LIN {X -0.159,Y -588.580,Z 1011.414,A 0.000,B 0.000,C 90.000,E1 110.536} C_DIS
LIN {X -0.262,Y -576.719,Z 1011.409,A 0.000,B 0.000,C 90.000,E1 109.577} C_DIS
LIN {X -0.071,Y -572.266,Z 1011.407,A 0.000,B 0.000,C 90.000,E1 109.214} C_DIS
LIN {X 0.230,Y -568.596,Z 1011.406,A 0.000,B 0.000,C 90.000,E1 108.960} C_DIS
LIN {X -0.107,Y -563.937,Z 1011.404,A 0.000,B 0.000,C 90.000,E1 108.725} C_DIS
LIN {X 0.068,Y -550.293,Z 1011.400,A 0.000,B 0.000,C 90.000,E1 108.000} C_DIS
LIN {X 0.171,Y -549.702,Z 1011.400,A 0.000,B 0.000,C 90.000,E1 107.946} C_DIS
LIN {X 0.114,Y -548.574,Z 1011.399,A 0.000,B 0.000,C 90.000,E1 107.819} C_DIS
LIN {X 0.072,Y -548.543,Z 1011.399,A 0.000,B 0.000,C 90.000,E1 107.819} C_DIS
LIN {X 0.076,Y -548.176,Z 1011.397,A 0.000,B 0.000,C 90.000,E1 107.511} C_DIS
LIN {X 0.119,Y -548.260,Z 1011.393,A 0.000,B 0.000,C 90.000,E1 106.804} C_DIS
LIN {X 0.030,Y -548.709,Z 1011.389,A 0.000,B 0.000,C 90.000,E1 105.969} C_DIS
LIN {X 0.074,Y -549.831,Z 1011.376,A 0.000,B 0.000,C 90.000,E1 103.716} C_DIS
LIN {X 0.056,Y -552.884,Z 1011.356,A 0.000,B 0.000,C 90.000,E1 100.074} C_DIS
LIN {X 0.060,Y -554.798,Z 1011.347,A 0.000,B 0.000,C 90.000,E1 98.398} C_DIS
LIN {X 0.114,Y -556.576,Z 1011.337,A 0.000,B 0.000,C 90.000,E1 96.720} C_DIS
LIN {X -0.128,Y -557.430,Z 1011.333,A 0.000,B 0.000,C 90.000,E1 95.910} C_DIS
LIN {X -0.220,Y -558.596,Z 1011.325,A 0.000,B 0.000,C 90.000,E1 94.531} C_DIS
LIN {X 0.262,Y -559.463,Z 1011.317,A 0.000,B 0.000,C 90.000,E1 93.094} C_DIS
LIN {X -0.033,Y -559.868,Z 1011.313,A 0.000,B 0.000,C 90.000,E1 92.293} C_DIS
LIN {X -0.023,Y -560.621,Z 1011.304,A 0.000,B 0.000,C 90.000,E1 90.630} C_DIS
LIN {X -0.009,Y -561.387,Z 1011.294,A 0.000,B 0.000,C 90.000,E1 88.969} C_DIS
LIN {X -0.164,Y -561.762,Z 1011.288,A 0.000,B 0.000,C 90.000,E1 87.879} C_DIS
LIN {X 0.253,Y -562.003,Z 1011.282,A 0.000,B 0.000,C 90.000,E1 86.731} C_DIS
LIN {X 0.100,Y -562.394,Z 1011.268,A 0.000,B 0.000,C 90.000,E1 84.261} C_DIS
LIN {X 0.005,Y -562.617,Z 1011.262,A 0.000,B 0.000,C 90.000,E1 83.166} C_DIS
LIN {X 0.214,Y -562.994,Z 1011.253,A 0.000,B 0.000,C 90.000,E1 81.489} C_DIS
LIN {X 0.027,Y -563.601,Z 1011.242,A 0.000,B 0.000,C 90.000,E1 79.577} C_DIS
LIN {X 0.059,Y -564.463,Z 1011.231,A 0.000,B 0.000,C 90.000,E1 77.645} C_DIS
LIN {X -0.086,Y -565.240,Z 1011.224,A 0.000,B 0.000,C 90.000,E1 76.284} C_DIS
LIN {X -0.261,Y -566.722,Z 1011.212,A 0.000,B 0.000,C 90.000,E1 74.102} C_DIS
LIN {X 0.119,Y -567.995,Z 1011.202,A 0.000,B 0.000,C 90.000,E1 72.417} C_DIS
LIN {X -0.006,Y -569.187,Z 1011.193,A 0.000,B 0.000,C 90.000,E1 70.786} C_DIS
LIN {X -0.082,Y -569.968,Z 1011.187,A 0.000,B 0.000,C 90.000,E1 69.699} C_DIS
LIN {X 0.010,Y -570.996,Z 1011.178,A 0.000,B 0.000,C 90.000,E1 68.050} C_DIS
LIN {X -0.367,Y -572.057,Z 1011.167,A 0.000,B 0.000,C 90.000,E1 66.177} C_DIS
LIN {X -0.319,Y -572.740,Z 1011.158,A 0.000,B 0.000,C 90.000,E1 64.537} C_DIS
LIN {X -0.007,Y -573.387,Z 1011.149,A 0.000,B 0.000,C 90.000,E1 62.871} C_DIS
LIN {X -0.193,Y -573.864,Z 1011.140,A 0.000,B 0.000,C 90.000,E1 61.257} C_DIS
LIN {X 0.064,Y -574.299,Z 1011.133,A 0.000,B 0.000,C 90.000,E1 59.871} C_DIS
LIN {X -0.165,Y -574.663,Z 1011.125,A 0.000,B 0.000,C 90.000,E1 58.535} C_DIS
LIN {X -0.083,Y -574.902,Z 1011.118,A 0.000,B 0.000,C 90.000,E1 57.168} C_DIS
LIN {X 0.005,Y -575.170,Z 1011.110,A 0.000,B 0.000,C 90.000,E1 55.801} C_DIS
LIN {X -0.384,Y -575.243,Z 1011.103,A 0.000,B 0.000,C 90.000,E1 54.482} C_DIS
LIN {X 0.216,Y -575.087,Z 1011.096,A 0.000,B 0.000,C 90.000,E1 53.336} C_DIS
LIN {X -0.140,Y -574.888,Z 1011.092,A 0.000,B 0.000,C 90.000,E1 52.557} C_DIS
LIN {X -0.001,Y -574.493,Z 1011.086,A 0.000,B 0.000,C 90.000,E1 51.457} C_DIS
LIN {X 0.134,Y -573.938,Z 1011.080,A 0.000,B 0.000,C 90.000,E1 50.356} C_DIS
LIN {X -0.182,Y -573.202,Z 1011.074,A 0.000,B 0.000,C 90.000,E1 49.299} C_DIS
LIN {X 0.300,Y -572.280,Z 1011.068,A 0.000,B 0.000,C 90.000,E1 48.162} C_DIS
LIN {X -0.167,Y -571.440,Z 1011.063,A 0.000,B 0.000,C 90.000,E1 47.391} C_DIS
LIN {X 0.162,Y -570.483,Z 1011.059,A 0.000,B 0.000,C 90.000,E1 46.539} C_DIS
LIN {X 0.368,Y -569.758,Z 1011.056,A 0.000,B 0.000,C 90.000,E1 45.972} C_DIS
LIN {X 0.056,Y -567.416,Z 1011.048,A 0.000,B 0.000,C 90.000,E1 44.636} C_DIS
LIN {X 0.021,Y -565.258,Z 1011.042,A 0.000,B 0.000,C 90.000,E1 43.542} C_DIS
LIN {X -0.198,Y -564.074,Z 1011.039,A 0.000,B 0.000,C 90.000,E1 43.014} C_DIS
LIN {X -0.271,Y -561.257,Z 1011.033,A 0.000,B 0.000,C 90.000,E1 41.919} C_DIS
LIN {X -0.140,Y -559.686,Z 1011.030,A 0.000,B 0.000,C 90.000,E1 41.353} C_DIS
LIN {X -0.309,Y -557.052,Z 1011.025,A 0.000,B 0.000,C 90.000,E1 40.539} C_DIS
LIN {X 0.281,Y -554.198,Z 1011.020,A 0.000,B 0.000,C 90.000,E1 39.644} C_DIS
LIN {X 0.060,Y -550.991,Z 1011.016,A 0.000,B 0.000,C 90.000,E1 38.830} C_DIS
LIN {X -0.196,Y -547.378,Z 1011.011,A 0.000,B 0.000,C 90.000,E1 38.016} C_DIS
LIN {X -0.064,Y -543.509,Z 1011.006,A 0.000,B 0.000,C 90.000,E1 37.156} C_DIS
LIN {X 0.045,Y -537.994,Z 1011.000,A 0.000,B 0.000,C 90.000,E1 36.011} C_DIS
LIN {X 0.068,Y -533.541,Z 1010.995,A 0.000,B 0.000,C 90.000,E1 35.152} C_DIS
LIN {X -0.247,Y -530.376,Z 1010.992,A 0.000,B 0.000,C 90.000,E1 34.612} C_DIS
LIN {X -0.037,Y -524.504,Z 1010.987,A 0.000,B 0.000,C 90.000,E1 33.579} C_DIS
LIN {X 0.150,Y -520.008,Z 1010.983,A 0.000,B 0.000,C 90.000,E1 32.832} C_DIS
LIN {X 0.030,Y -516.170,Z 1010.979,A 0.000,B 0.000,C 90.000,E1 32.260} C_DIS
LIN {X 0.042,Y -512.089,Z 1010.976,A 0.000,B 0.000,C 90.000,E1 31.671} C_DIS
LIN {X 0.030,Y -507.722,Z 1010.973,A 0.000,B 0.000,C 90.000,E1 31.082} C_DIS
LIN {X 0.054,Y -501.796,Z 1010.969,A 0.000,B 0.000,C 90.000,E1 30.335} C_DIS
LIN {X 0.046,Y -495.398,Z 1010.964,A 0.000,B 0.000,C 90.000,E1 29.589} C_DIS
LIN {X 0.004,Y -490.028,Z 1010.961,A 0.000,B 0.000,C 90.000,E1 28.999} C_DIS
LIN {X -0.134,Y -480.140,Z 1010.956,A 0.000,B 0.000,C 90.000,E1 28.025} C_DIS
LIN {X 0.044,Y -472.911,Z 1010.952,A 0.000,B 0.000,C 90.000,E1 27.308} C_DIS
LIN {X 0.131,Y -464.219,Z 1010.947,A 0.000,B 0.000,C 90.000,E1 26.488} C_DIS
LIN {X 0.025,Y -456.800,Z 1010.944,A 0.000,B 0.000,C 90.000,E1 25.848} C_DIS
LIN {X -0.094,Y -446.071,Z 1010.939,A 0.000,B 0.000,C 90.000,E1 24.951} C_DIS
LIN {X -0.172,Y -428.098,Z 1010.930,A 0.000,B 0.000,C 90.000,E1 23.387} C_DIS
LIN {X -0.101,Y -422.103,Z 1010.927,A 0.000,B 0.000,C 90.000,E1 22.823} C_DIS
LIN {X -0.068,Y -408.351,Z 1010.919,A 0.000,B 0.000,C 90.000,E1 21.408} C_DIS
LIN {X 0.103,Y -399.893,Z 1010.914,A 0.000,B 0.000,C 90.000,E1 20.429} C_DIS
LIN {X -0.029,Y -396.273,Z 1010.911,A 0.000,B 0.000,C 90.000,E1 19.993} C_DIS
LIN {X 0.148,Y -393.953,Z 1010.909,A 0.000,B 0.000,C 90.000,E1 19.577} C_DIS
LIN {X -0.191,Y -393.063,Z 1010.908,A 0.000,B 0.000,C 90.000,E1 19.450} C_DIS
LIN {X 0.130,Y -391.491,Z 1010.906,A 0.000,B 0.000,C 90.000,E1 18.960} C_DIS
LIN {X -0.058,Y -390.916,Z 1010.903,A 0.000,B 0.000,C 90.000,E1 18.544} C_DIS
LIN {X -0.011,Y -390.829,Z 1010.901,A 0.000,B 0.000,C 90.000,E1 18.181} C_DIS
LIN {X 0.033,Y -390.836,Z 1010.899,A 0.000,B 0.000,C 90.000,E1 17.819} C_DIS
LIN {X 0.185,Y -393.306,Z 1010.883,A 0.000,B 0.000,C 90.000,E1 14.954} C_DIS
LIN {X 0.162,Y -397.687,Z 1010.864,A 0.000,B 0.000,C 90.000,E1 11.422} C_DIS
LIN {X 0.087,Y -402.785,Z 1010.846,A 0.000,B 0.000,C 90.000,E1 8.276} C_DIS
LIN {X -0.040,Y -408.148,Z 1010.831,A 0.000,B 0.000,C 90.000,E1 5.511} C_DIS
LIN {X -0.042,Y -412.638,Z 1010.819,A 0.000,B 0.000,C 90.000,E1 3.440} C_DIS
LIN {X -0.010,Y -415.871,Z 1010.812,A 0.000,B 0.000,C 90.000,E1 2.064} C_DIS
LIN {X 0.024,Y -417.553,Z 1010.809,A 0.000,B 0.000,C 90.000,E1 1.547} C_DIS
LIN {X 0.134,Y -419.888,Z 1010.806,A 0.000,B 0.000,C 90.000,E1 1.031} C_DIS
LIN {X 0.165,Y -422.361,Z 1010.804,A 0.000,B 0.000,C 90.000,E1 0.688} C_DIS
LIN {X 0.184,Y -423.875,Z 1010.803,A 0.000,B 0.000,C 90.000,E1 0.516} C_DIS
LIN {X 0.059,Y -427.432,Z 1010.801,A 0.000,B 0.000,C 90.000,E1 0.229} C_DIS
LIN {X 0.165,Y -434.773,Z 1010.799,A 0.000,B 0.000,C 90.000,E1 359.771} C_DIS
LIN {X 0.007,Y -443.154,Z 1010.796,A 0.000,B 0.000,C 90.000,E1 359.312} C_DIS
LIN {X -0.039,Y -459.882,Z 1010.791,A 0.000,B 0.000,C 90.000,E1 358.339} C_DIS
LIN {X -0.089,Y -479.668,Z 1010.784,A 0.000,B 0.000,C 90.000,E1 357.192} C_DIS
LIN {X -0.222,Y -487.813,Z 1010.782,A 0.000,B 0.000,C 90.000,E1 356.731} C_DIS
LIN {X 0.114,Y -502.438,Z 1010.777,A 0.000,B 0.000,C 90.000,E1 355.812} C_DIS
LIN {X 0.211,Y -510.388,Z 1010.774,A 0.000,B 0.000,C 90.000,E1 355.298} C_DIS
LIN {X 0.103,Y -516.478,Z 1010.772,A 0.000,B 0.000,C 90.000,E1 354.894} C_DIS
LIN {X -0.247,Y -524.067,Z 1010.769,A 0.000,B 0.000,C 90.000,E1 354.375} C_DIS
LIN {X 0.169,Y -531.406,Z 1010.765,A 0.000,B 0.000,C 90.000,E1 353.742} C_DIS
LIN {X -0.197,Y -539.633,Z 1010.761,A 0.000,B 0.000,C 90.000,E1 353.053} C_DIS
LIN {X 0.217,Y -546.269,Z 1010.758,A 0.000,B 0.000,C 90.000,E1 352.356} C_DIS
LIN {X 0.030,Y -551.375,Z 1010.755,A 0.000,B 0.000,C 90.000,E1 351.837} C_DIS
LIN {X 0.311,Y -556.103,Z 1010.752,A 0.000,B 0.000,C 90.000,E1 351.254} C_DIS
LIN {X -0.315,Y -561.492,Z 1010.748,A 0.000,B 0.000,C 90.000,E1 350.622} C_DIS
LIN {X -0.010,Y -565.410,Z 1010.745,A 0.000,B 0.000,C 90.000,E1 350.038} C_DIS
LIN {X -0.230,Y -568.963,Z 1010.742,A 0.000,B 0.000,C 90.000,E1 349.511} C_DIS
LIN {X -0.145,Y -575.362,Z 1010.736,A 0.000,B 0.000,C 90.000,E1 348.409} C_DIS
LIN {X 0.154,Y -579.035,Z 1010.732,A 0.000,B 0.000,C 90.000,E1 347.701} C_DIS
LIN {X 0.260,Y -583.056,Z 1010.727,A 0.000,B 0.000,C 90.000,E1 346.881} C_DIS
LIN {X 0.082,Y -588.192,Z 1010.721,A 0.000,B 0.000,C 90.000,E1 345.825} C_DIS
LIN {X 0.347,Y -592.388,Z 1010.716,A 0.000,B 0.000,C 90.000,E1 344.866} C_DIS
LIN {X -0.133,Y -597.005,Z 1010.710,A 0.000,B 0.000,C 90.000,E1 343.850} C_DIS
LIN {X -0.266,Y -602.405,Z 1010.703,A 0.000,B 0.000,C 90.000,E1 342.543} C_DIS
LIN {X -0.138,Y -607.443,Z 1010.696,A 0.000,B 0.000,C 90.000,E1 341.221} C_DIS
LIN {X 0.025,Y -610.304,Z 1010.691,A 0.000,B 0.000,C 90.000,E1 340.423} C_DIS
LIN {X 0.012,Y -612.929,Z 1010.687,A 0.000,B 0.000,C 90.000,E1 339.645} C_DIS
LIN {X 0.167,Y -616.982,Z 1010.680,A 0.000,B 0.000,C 90.000,E1 338.337} C_DIS
LIN {X 0.156,Y -621.442,Z 1010.671,A 0.000,B 0.000,C 90.000,E1 336.794} C_DIS
LIN {X -0.107,Y -624.118,Z 1010.666,A 0.000,B 0.000,C 90.000,E1 335.793} C_DIS
LIN {X -0.339,Y -626.594,Z 1010.660,A 0.000,B 0.000,C 90.000,E1 334.793} C_DIS
LIN {X -0.250,Y -629.500,Z 1010.653,A 0.000,B 0.000,C 90.000,E1 333.512} C_DIS
LIN {X -0.171,Y -630.936,Z 1010.649,A 0.000,B 0.000,C 90.000,E1 332.743} C_DIS
LIN {X -0.048,Y -632.856,Z 1010.643,A 0.000,B 0.000,C 90.000,E1 331.719} C_DIS
LIN {X -0.077,Y -635.383,Z 1010.634,A 0.000,B 0.000,C 90.000,E1 330.205} C_DIS
LIN {X -0.185,Y -636.529,Z 1010.630,A 0.000,B 0.000,C 90.000,E1 329.459} C_DIS
LIN {X -0.189,Y -638.190,Z 1010.623,A 0.000,B 0.000,C 90.000,E1 328.201} C_DIS
LIN {X 0.125,Y -639.381,Z 1010.618,A 0.000,B 0.000,C 90.000,E1 327.168} C_DIS
LIN {X -0.031,Y -640.710,Z 1010.611,A 0.000,B 0.000,C 90.000,E1 325.928} C_DIS
LIN {X 0.319,Y -641.463,Z 1010.605,A 0.000,B 0.000,C 90.000,E1 324.895} C_DIS
LIN {X 0.152,Y -642.056,Z 1010.600,A 0.000,B 0.000,C 90.000,E1 323.909} C_DIS
LIN {X -0.116,Y -642.558,Z 1010.593,A 0.000,B 0.000,C 90.000,E1 322.683} C_DIS
LIN {X -0.052,Y -643.140,Z 1010.582,A 0.000,B 0.000,C 90.000,E1 320.678} C_DIS
LIN {X 0.171,Y -644.162,Z 1010.568,A 0.000,B 0.000,C 90.000,E1 318.162} C_DIS
LIN {X -0.161,Y -644.774,Z 1010.561,A 0.000,B 0.000,C 90.000,E1 316.944} C_DIS
LIN {X 0.333,Y -645.537,Z 1010.552,A 0.000,B 0.000,C 90.000,E1 315.405} C_DIS
LIN {X -0.197,Y -646.759,Z 1010.541,A 0.000,B 0.000,C 90.000,E1 313.461} C_DIS
LIN {X -0.050,Y -647.516,Z 1010.534,A 0.000,B 0.000,C 90.000,E1 312.204} C_DIS
LIN {X 0.031,Y -648.357,Z 1010.525,A 0.000,B 0.000,C 90.000,E1 310.458} C_DIS
LIN {X -0.215,Y -648.925,Z 1010.517,A 0.000,B 0.000,C 90.000,E1 308.991} C_DIS
LIN {X -0.049,Y -649.465,Z 1010.508,A 0.000,B 0.000,C 90.000,E1 307.488} C_DIS
LIN {X 0.314,Y -649.765,Z 1010.501,A 0.000,B 0.000,C 90.000,E1 306.217} C_DIS
LIN {X -0.218,Y -649.975,Z 1010.495,A 0.000,B 0.000,C 90.000,E1 305.025} C_DIS
LIN {X -0.056,Y -651.341,Z 1010.475,A 0.000,B 0.000,C 90.000,E1 301.544} C_DIS
LIN {X -0.005,Y -653.853,Z 1010.460,A 0.000,B 0.000,C 90.000,E1 298.821} C_DIS
LIN {X -0.152,Y -656.585,Z 1010.448,A 0.000,B 0.000,C 90.000,E1 296.616} C_DIS
LIN {X 0.326,Y -657.849,Z 1010.442,A 0.000,B 0.000,C 90.000,E1 295.591} C_DIS
LIN {X -0.058,Y -658.955,Z 1010.437,A 0.000,B 0.000,C 90.000,E1 294.643} C_DIS
LIN {X 0.172,Y -659.664,Z 1010.431,A 0.000,B 0.000,C 90.000,E1 293.643} C_DIS
LIN {X 0.162,Y -659.900,Z 1010.429,A 0.000,B 0.000,C 90.000,E1 293.153} C_DIS
LIN {X -0.204,Y -660.124,Z 1010.423,A 0.000,B 0.000,C 90.000,E1 292.206} C_DIS
LIN {X -0.208,Y -659.893,Z 1010.421,A 0.000,B 0.000,C 90.000,E1 291.716} C_DIS
LIN {X -0.089,Y -659.582,Z 1010.419,A 0.000,B 0.000,C 90.000,E1 291.461} C_DIS
LIN {X -0.095,Y -658.617,Z 1010.417,A 0.000,B 0.000,C 90.000,E1 290.972} C_DIS
LIN {X -0.216,Y -657.599,Z 1010.415,A 0.000,B 0.000,C 90.000,E1 290.737} C_DIS
LIN {X -0.230,Y -655.013,Z 1010.412,A 0.000,B 0.000,C 90.000,E1 290.248} C_DIS
LIN {X -0.181,Y -653.942,Z 1010.412,A 0.000,B 0.000,C 90.000,E1 290.120} C_DIS
LIN {X 0.247,Y -648.184,Z 1010.409,A 0.000,B 0.000,C 90.000,E1 289.631} C_DIS
LIN {X -0.342,Y -646.603,Z 1010.409,A 0.000,B 0.000,C 90.000,E1 289.577} C_DIS
LIN {X 0.314,Y -640.242,Z 1010.407,A 0.000,B 0.000,C 90.000,E1 289.141} C_DIS
LIN {X -0.269,Y -633.177,Z 1010.405,A 0.000,B 0.000,C 90.000,E1 288.852} C_DIS
LIN {X -0.152,Y -629.797,Z 1010.404,A 0.000,B 0.000,C 90.000,E1 288.652} C_DIS
LIN {X -0.201,Y -629.765,Z 1010.404,A 0.000,B 0.000,C 90.000,E1 288.652} C_DIS
LIN {X 0.325,Y -628.643,Z 1010.403,A 0.000,B 0.000,C 90.000,E1 288.417} C_DIS
LIN {X 0.281,Y -628.644,Z 1010.403,A 0.000,B 0.000,C 90.000,E1 288.417} C_DIS
LIN {X -0.188,Y -632.132,Z 1010.399,A 0.000,B 0.000,C 90.000,E1 287.873} C_DIS
LIN {X -0.039,Y -635.307,Z 1010.397,A 0.000,B 0.000,C 90.000,E1 287.402} C_DIS
LIN {X -0.219,Y -637.821,Z 1010.395,A 0.000,B 0.000,C 90.000,E1 287.040} C_DIS
LIN {X -0.216,Y -638.747,Z 1010.394,A 0.000,B 0.000,C 90.000,E1 286.913} C_DIS
LIN {X 0.071,Y -642.338,Z 1010.390,A 0.000,B 0.000,C 90.000,E1 286.260} C_DIS
LIN {X 0.080,Y -643.126,Z 1010.390,A 0.000,B 0.000,C 90.000,E1 286.134} C_DIS
LIN {X 0.244,Y -646.733,Z 1010.386,A 0.000,B 0.000,C 90.000,E1 285.371} C_DIS
LIN {X -0.039,Y -648.542,Z 1010.383,A 0.000,B 0.000,C 90.000,E1 284.898} C_DIS
LIN {X -0.148,Y -650.055,Z 1010.380,A 0.000,B 0.000,C 90.000,E1 284.411} C_DIS
LIN {X 0.348,Y -650.753,Z 1010.379,A 0.000,B 0.000,C 90.000,E1 284.120} C_DIS
LIN {X 0.088,Y -651.781,Z 1010.376,A 0.000,B 0.000,C 90.000,E1 283.647} C_DIS
LIN {X -0.165,Y -652.511,Z 1010.373,A 0.000,B 0.000,C 90.000,E1 283.175} C_DIS
LIN {X 0.098,Y -653.160,Z 1010.369,A 0.000,B 0.000,C 90.000,E1 282.411} C_DIS
LIN {X 0.233,Y -653.263,Z 1010.365,A 0.000,B 0.000,C 90.000,E1 281.658} C_DIS
LIN {X -0.012,Y -653.008,Z 1010.362,A 0.000,B 0.000,C 90.000,E1 281.186} C_DIS
LIN {X -0.263,Y -652.505,Z 1010.359,A 0.000,B 0.000,C 90.000,E1 280.715} C_DIS
LIN {X 0.005,Y -651.696,Z 1010.357,A 0.000,B 0.000,C 90.000,E1 280.197} C_DIS
LIN {X -0.258,Y -650.574,Z 1010.354,A 0.000,B 0.000,C 90.000,E1 279.726} C_DIS
LIN {X 0.140,Y -649.971,Z 1010.353,A 0.000,B 0.000,C 90.000,E1 279.443} C_DIS
LIN {X -0.137,Y -648.356,Z 1010.350,A 0.000,B 0.000,C 90.000,E1 278.973} C_DIS
LIN {X 0.113,Y -646.327,Z 1010.347,A 0.000,B 0.000,C 90.000,E1 278.454} C_DIS
LIN {X -0.285,Y -643.886,Z 1010.344,A 0.000,B 0.000,C 90.000,E1 277.992} C_DIS
LIN {X 0.191,Y -642.464,Z 1010.343,A 0.000,B 0.000,C 90.000,E1 277.701} C_DIS
LIN {X -0.234,Y -639.084,Z 1010.340,A 0.000,B 0.000,C 90.000,E1 277.239} C_DIS
LIN {X -0.045,Y -635.183,Z 1010.337,A 0.000,B 0.000,C 90.000,E1 276.720} C_DIS
LIN {X -0.006,Y -629.271,Z 1010.334,A 0.000,B 0.000,C 90.000,E1 276.087} C_DIS
LIN {X 0.272,Y -624.170,Z 1010.331,A 0.000,B 0.000,C 90.000,E1 275.568} C_DIS
LIN {X 0.152,Y -618.794,Z 1010.328,A 0.000,B 0.000,C 90.000,E1 275.106} C_DIS
LIN {X -0.288,Y -612.957,Z 1010.326,A 0.000,B 0.000,C 90.000,E1 274.702} C_DIS
LIN {X 0.233,Y -606.741,Z 1010.324,A 0.000,B 0.000,C 90.000,E1 274.245} C_DIS
LIN {X -0.111,Y -600.202,Z 1010.322,A 0.000,B 0.000,C 90.000,E1 273.898} C_DIS
LIN {X 0.097,Y -594.950,Z 1010.320,A 0.000,B 0.000,C 90.000,E1 273.612} C_DIS
LIN {X 0.213,Y -591.632,Z 1010.319,A 0.000,B 0.000,C 90.000,E1 273.440} C_DIS
LIN {X -0.276,Y -585.600,Z 1010.318,A 0.000,B 0.000,C 90.000,E1 273.269} C_DIS
LIN {X -0.195,Y -577.962,Z 1010.317,A 0.000,B 0.000,C 90.000,E1 273.037} C_DIS
LIN {X 0.186,Y -572.428,Z 1010.316,A 0.000,B 0.000,C 90.000,E1 272.865} C_DIS
LIN {X 0.157,Y -565.651,Z 1010.315,A 0.000,B 0.000,C 90.000,E1 272.751} C_DIS
LIN {X 0.189,Y -558.341,Z 1010.315,A 0.000,B 0.000,C 90.000,E1 272.694} C_DIS
LIN {X 0.139,Y -543.327,Z 1010.315,A 0.000,B 0.000,C 90.000,E1 272.694} C_DIS
LIN {X 0.079,Y -542.751,Z 1010.313,A 0.000,B 0.000,C 90.000,E1 272.407} C_DIS
LIN {X 0.216,Y -542.125,Z 1010.310,A 0.000,B 0.000,C 90.000,E1 271.835} C_DIS
LIN {X -0.132,Y -540.870,Z 1010.299,A 0.000,B 0.000,C 90.000,E1 269.885} C_DIS
LIN {X -0.025,Y -539.956,Z 1010.291,A 0.000,B 0.000,C 90.000,E1 268.453} C_DIS
LIN {X 0.045,Y -539.358,Z 1010.287,A 0.000,B 0.000,C 90.000,E1 267.593} C_DIS
LIN {X 0.186,Y -537.812,Z 1010.276,A 0.000,B 0.000,C 90.000,E1 265.584} C_DIS
LIN {X -0.203,Y -536.488,Z 1010.266,A 0.000,B 0.000,C 90.000,E1 263.913} C_DIS
LIN {X -0.072,Y -535.236,Z 1010.258,A 0.000,B 0.000,C 90.000,E1 262.470} C_DIS
LIN {X 0.027,Y -533.831,Z 1010.250,A 0.000,B 0.000,C 90.000,E1 261.027} C_DIS
LIN {X 0.220,Y -532.615,Z 1010.244,A 0.000,B 0.000,C 90.000,E1 259.859} C_DIS
LIN {X -0.066,Y -530.067,Z 1010.231,A 0.000,B 0.000,C 90.000,E1 257.589} C_DIS
LIN {X 0.218,Y -528.545,Z 1010.223,A 0.000,B 0.000,C 90.000,E1 256.117} C_DIS
LIN {X 0.134,Y -526.260,Z 1010.212,A 0.000,B 0.000,C 90.000,E1 254.102} C_DIS
LIN {X -0.028,Y -524.699,Z 1010.204,A 0.000,B 0.000,C 90.000,E1 252.670} C_DIS
LIN {X -0.060,Y -523.087,Z 1010.196,A 0.000,B 0.000,C 90.000,E1 251.221} C_DIS
LIN {X 0.054,Y -521.211,Z 1010.188,A 0.000,B 0.000,C 90.000,E1 249.752} C_DIS
LIN {X -0.054,Y -518.588,Z 1010.176,A 0.000,B 0.000,C 90.000,E1 247.720} C_DIS
LIN {X 0.036,Y -516.984,Z 1010.170,A 0.000,B 0.000,C 90.000,E1 246.538} C_DIS
LIN {X -0.244,Y -514.866,Z 1010.162,A 0.000,B 0.000,C 90.000,E1 245.101} C_DIS
LIN {X -0.121,Y -513.572,Z 1010.157,A 0.000,B 0.000,C 90.000,E1 244.204} C_DIS
LIN {X -0.250,Y -511.196,Z 1010.148,A 0.000,B 0.000,C 90.000,E1 242.743} C_DIS
LIN {X 0.132,Y -508.341,Z 1010.139,A 0.000,B 0.000,C 90.000,E1 240.923} C_DIS
LIN {X -0.064,Y -505.758,Z 1010.130,A 0.000,B 0.000,C 90.000,E1 239.459} C_DIS
LIN {X 0.194,Y -504.107,Z 1010.125,A 0.000,B 0.000,C 90.000,E1 238.535} C_DIS
LIN {X 0.181,Y -501.177,Z 1010.117,A 0.000,B 0.000,C 90.000,E1 237.041} C_DIS
LIN {X -0.175,Y -498.568,Z 1010.110,A 0.000,B 0.000,C 90.000,E1 235.881} C_DIS
LIN {X -0.156,Y -496.584,Z 1010.105,A 0.000,B 0.000,C 90.000,E1 234.975} C_DIS
LIN {X -0.008,Y -493.625,Z 1010.099,A 0.000,B 0.000,C 90.000,E1 233.749} C_DIS
LIN {X -0.196,Y -490.682,Z 1010.092,A 0.000,B 0.000,C 90.000,E1 232.557} C_DIS
LIN {X -0.022,Y -485.613,Z 1010.080,A 0.000,B 0.000,C 90.000,E1 230.400} C_DIS
LIN {X 0.081,Y -482.059,Z 1010.072,A 0.000,B 0.000,C 90.000,E1 228.852} C_DIS
LIN {X 0.195,Y -475.944,Z 1010.056,A 0.000,B 0.000,C 90.000,E1 226.053} C_DIS
LIN {X 0.235,Y -471.520,Z 1010.044,A 0.000,B 0.000,C 90.000,E1 223.866} C_DIS
LIN {X 0.166,Y -466.861,Z 1010.032,A 0.000,B 0.000,C 90.000,E1 221.676} C_DIS
LIN {X 0.211,Y -463.462,Z 1010.023,A 0.000,B 0.000,C 90.000,E1 220.092} C_DIS
LIN {X 0.153,Y -460.594,Z 1010.016,A 0.000,B 0.000,C 90.000,E1 218.830} C_DIS
LIN {X -0.119,Y -456.352,Z 1010.005,A 0.000,B 0.000,C 90.000,E1 216.950} C_DIS
LIN {X -0.124,Y -452.141,Z 1009.995,A 0.000,B 0.000,C 90.000,E1 215.025} C_DIS
LIN {X 0.025,Y -446.480,Z 1009.980,A 0.000,B 0.000,C 90.000,E1 212.418} C_DIS
LIN {X 0.081,Y -441.507,Z 1009.967,A 0.000,B 0.000,C 90.000,E1 210.129} C_DIS
LIN {X 0.006,Y -439.348,Z 1009.962,A 0.000,B 0.000,C 90.000,E1 209.155} C_DIS
LIN {X -0.012,Y -434.779,Z 1009.951,A 0.000,B 0.000,C 90.000,E1 207.180} C_DIS
LIN {X -0.151,Y -431.069,Z 1009.942,A 0.000,B 0.000,C 90.000,E1 205.540} C_DIS
LIN {X 0.213,Y -427.325,Z 1009.933,A 0.000,B 0.000,C 90.000,E1 203.823} C_DIS
LIN {X 0.126,Y -422.103,Z 1009.919,A 0.000,B 0.000,C 90.000,E1 201.482} C_DIS
LIN {X -0.100,Y -417.314,Z 1009.906,A 0.000,B 0.000,C 90.000,E1 199.141} C_DIS
LIN {X 0.044,Y -412.927,Z 1009.893,A 0.000,B 0.000,C 90.000,E1 196.732} C_DIS
LIN {X -0.168,Y -408.922,Z 1009.880,A 0.000,B 0.000,C 90.000,E1 194.356} C_DIS
LIN {X 0.114,Y -405.296,Z 1009.866,A 0.000,B 0.000,C 90.000,E1 191.895} C_DIS
LIN {X -0.172,Y -402.664,Z 1009.855,A 0.000,B 0.000,C 90.000,E1 189.849} C_DIS
LIN {X -0.174,Y -402.053,Z 1009.851,A 0.000,B 0.000,C 90.000,E1 189.151} C_DIS
LIN {X -0.182,Y -401.886,Z 1009.847,A 0.000,B 0.000,C 90.000,E1 188.454} C_DIS
LIN {X -0.194,Y -402.215,Z 1009.843,A 0.000,B 0.000,C 90.000,E1 187.757} C_DIS
LIN {X 0.141,Y -403.219,Z 1009.839,A 0.000,B 0.000,C 90.000,E1 187.011} C_DIS
LIN {X 0.159,Y -404.411,Z 1009.836,A 0.000,B 0.000,C 90.000,E1 186.486} C_DIS
LIN {X -0.152,Y -407.346,Z 1009.832,A 0.000,B 0.000,C 90.000,E1 185.796} C_DIS
LIN {X -0.146,Y -409.187,Z 1009.830,A 0.000,B 0.000,C 90.000,E1 185.448} C_DIS
LIN {X -0.180,Y -412.261,Z 1009.827,A 0.000,B 0.000,C 90.000,E1 184.935} C_DIS
LIN {X 0.187,Y -415.702,Z 1009.825,A 0.000,B 0.000,C 90.000,E1 184.416} C_DIS
LIN {X 0.200,Y -428.181,Z 1009.816,A 0.000,B 0.000,C 90.000,E1 182.922} C_DIS
LIN {X 0.012,Y -436.600,Z 1009.811,A 0.000,B 0.000,C 90.000,E1 182.007} C_DIS
LIN {X -0.167,Y -446.138,Z 1009.805,A 0.000,B 0.000,C 90.000,E1 180.917} C_DIS
LIN {X 0.161,Y -455.560,Z 1009.799,A 0.000,B 0.000,C 90.000,E1 179.771} C_DIS
LIN {X 0.088,Y -463.361,Z 1009.794,A 0.000,B 0.000,C 90.000,E1 178.854} C_DIS
LIN {X 0.202,Y -469.855,Z 1009.789,A 0.000,B 0.000,C 90.000,E1 178.051} C_DIS
LIN {X 0.146,Y -478.630,Z 1009.783,A 0.000,B 0.000,C 90.000,E1 176.963} C_DIS
LIN {X -0.226,Y -482.138,Z 1009.781,A 0.000,B 0.000,C 90.000,E1 176.560} C_DIS
LIN {X -0.092,Y -486.756,Z 1009.777,A 0.000,B 0.000,C 90.000,E1 175.927} C_DIS
LIN {X -0.246,Y -495.535,Z 1009.771,A 0.000,B 0.000,C 90.000,E1 174.723} C_DIS
LIN {X -0.055,Y -503.529,Z 1009.764,A 0.000,B 0.000,C 90.000,E1 173.514} C_DIS
LIN {X -0.249,Y -511.268,Z 1009.757,A 0.000,B 0.000,C 90.000,E1 172.356} C_DIS
LIN {X -0.138,Y -517.755,Z 1009.752,A 0.000,B 0.000,C 90.000,E1 171.319} C_DIS
LIN {X 0.072,Y -527.246,Z 1009.743,A 0.000,B 0.000,C 90.000,E1 169.690} C_DIS
LIN {X 0.142,Y -536.544,Z 1009.734,A 0.000,B 0.000,C 90.000,E1 168.117} C_DIS
LIN {X -0.093,Y -545.559,Z 1009.725,A 0.000,B 0.000,C 90.000,E1 166.589} C_DIS
LIN {X 0.262,Y -555.100,Z 1009.716,A 0.000,B 0.000,C 90.000,E1 164.866} C_DIS
LIN {X -0.023,Y -560.425,Z 1009.711,A 0.000,B 0.000,C 90.000,E1 163.921} C_DIS
LIN {X -0.204,Y -566.237,Z 1009.705,A 0.000,B 0.000,C 90.000,E1 162.834} C_DIS
LIN {X 0.066,Y -571.839,Z 1009.698,A 0.000,B 0.000,C 90.000,E1 161.710} C_DIS
LIN {X -0.137,Y -575.954,Z 1009.694,A 0.000,B 0.000,C 90.000,E1 160.913} C_DIS
LIN {X -0.182,Y -581.717,Z 1009.687,A 0.000,B 0.000,C 90.000,E1 159.699} C_DIS
LIN {X 0.133,Y -586.580,Z 1009.681,A 0.000,B 0.000,C 90.000,E1 158.592} C_DIS
LIN {X -0.034,Y -591.112,Z 1009.675,A 0.000,B 0.000,C 90.000,E1 157.539} C_DIS
LIN {X -0.143,Y -595.323,Z 1009.669,A 0.000,B 0.000,C 90.000,E1 156.485} C_DIS
LIN {X 0.218,Y -597.338,Z 1009.666,A 0.000,B 0.000,C 90.000,E1 155.921} C_DIS
LIN {X -0.106,Y -600.991,Z 1009.661,A 0.000,B 0.000,C 90.000,E1 154.897} C_DIS
LIN {X -0.097,Y -604.322,Z 1009.655,A 0.000,B 0.000,C 90.000,E1 153.845} C_DIS
LIN {X -0.053,Y -607.431,Z 1009.649,A 0.000,B 0.000,C 90.000,E1 152.794} C_DIS
LIN {X -0.322,Y -611.868,Z 1009.640,A 0.000,B 0.000,C 90.000,E1 151.257} C_DIS
LIN {X -0.167,Y -614.725,Z 1009.634,A 0.000,B 0.000,C 90.000,E1 150.205} C_DIS
LIN {X -0.233,Y -618.884,Z 1009.626,A 0.000,B 0.000,C 90.000,E1 148.663} C_DIS
LIN {X -0.216,Y -622.939,Z 1009.617,A 0.000,B 0.000,C 90.000,E1 147.120} C_DIS
LIN {X 0.041,Y -627.626,Z 1009.607,A 0.000,B 0.000,C 90.000,E1 145.308} C_DIS
LIN {X 0.050,Y -631.630,Z 1009.599,A 0.000,B 0.000,C 90.000,E1 143.783} C_DIS
LIN {X -0.383,Y -634.920,Z 1009.592,A 0.000,B 0.000,C 90.000,E1 142.557} C_DIS
LIN {X 0.024,Y -638.840,Z 1009.583,A 0.000,B 0.000,C 90.000,E1 141.009} C_DIS
LIN {X 0.026,Y -642.641,Z 1009.575,A 0.000,B 0.000,C 90.000,E1 139.504} C_DIS
LIN {X 0.249,Y -645.132,Z 1009.570,A 0.000,B 0.000,C 90.000,E1 138.485} C_DIS
LIN {X -0.034,Y -647.664,Z 1009.564,A 0.000,B 0.000,C 90.000,E1 137.514} C_DIS
LIN {X -0.033,Y -653.693,Z 1009.552,A 0.000,B 0.000,C 90.000,E1 135.283} C_DIS
LIN {X -0.353,Y -661.246,Z 1009.538,A 0.000,B 0.000,C 90.000,E1 132.852} C_DIS
LIN {X 0.037,Y -666.002,Z 1009.530,A 0.000,B 0.000,C 90.000,E1 131.353} C_DIS
LIN {X 0.148,Y -670.627,Z 1009.522,A 0.000,B 0.000,C 90.000,E1 129.886} C_DIS
LIN {X 0.256,Y -674.200,Z 1009.515,A 0.000,B 0.000,C 90.000,E1 128.669} C_DIS
LIN {X -0.429,Y -677.664,Z 1009.508,A 0.000,B 0.000,C 90.000,E1 127.523} C_DIS
LIN {X -0.106,Y -680.995,Z 1009.502,A 0.000,B 0.000,C 90.000,E1 126.297} C_DIS
LIN {X -0.121,Y -684.893,Z 1009.494,A 0.000,B 0.000,C 90.000,E1 124.865} C_DIS
LIN {X -0.108,Y -687.414,Z 1009.488,A 0.000,B 0.000,C 90.000,E1 123.913} C_DIS
LIN {X 0.312,Y -689.241,Z 1009.484,A 0.000,B 0.000,C 90.000,E1 123.166} C_DIS
LIN {X -0.095,Y -693.402,Z 1009.475,A 0.000,B 0.000,C 90.000,E1 121.544} C_DIS
LIN {X 0.033,Y -695.735,Z 1009.470,A 0.000,B 0.000,C 90.000,E1 120.590} C_DIS
LIN {X -0.169,Y -697.719,Z 1009.465,A 0.000,B 0.000,C 90.000,E1 119.667} C_DIS
LIN {X 0.266,Y -699.301,Z 1009.460,A 0.000,B 0.000,C 90.000,E1 118.693} C_DIS
LIN {X -0.164,Y -700.269,Z 1009.456,A 0.000,B 0.000,C 90.000,E1 118.025} C_DIS
LIN {X 0.378,Y -700.744,Z 1009.453,A 0.000,B 0.000,C 90.000,E1 117.513} C_DIS
LIN {X 0.077,Y -702.241,Z 1009.443,A 0.000,B 0.000,C 90.000,E1 115.668} C_DIS
LIN {X -0.376,Y -702.886,Z 1009.438,A 0.000,B 0.000,C 90.000,E1 114.771} C_DIS
LIN {X 0.182,Y -702.947,Z 1009.435,A 0.000,B 0.000,C 90.000,E1 114.259} C_DIS
LIN {X 0.173,Y -702.802,Z 1009.434,A 0.000,B 0.000,C 90.000,E1 114.027} C_DIS
LIN {X 0.085,Y -702.062,Z 1009.431,A 0.000,B 0.000,C 90.000,E1 113.567} C_DIS
LIN {X 0.081,Y -701.260,Z 1009.430,A 0.000,B 0.000,C 90.000,E1 113.334} C_DIS
LIN {X 0.353,Y -700.222,Z 1009.428,A 0.000,B 0.000,C 90.000,E1 113.078} C_DIS
LIN {X -0.295,Y -699.036,Z 1009.427,A 0.000,B 0.000,C 90.000,E1 112.898} C_DIS
LIN {X -0.162,Y -698.192,Z 1009.426,A 0.000,B 0.000,C 90.000,E1 112.770} C_DIS
LIN {X -0.030,Y -696.938,Z 1009.426,A 0.000,B 0.000,C 90.000,E1 112.642} C_DIS
LIN {X 0.187,Y -690.637,Z 1009.424,A 0.000,B 0.000,C 90.000,E1 112.206} C_DIS
LIN {X -0.300,Y -688.644,Z 1009.423,A 0.000,B 0.000,C 90.000,E1 112.153} C_DIS
LIN {X 0.064,Y -683.849,Z 1009.422,A 0.000,B 0.000,C 90.000,E1 111.972} C_DIS
LIN {X 0.183,Y -675.272,Z 1009.422,A 0.000,B 0.000,C 90.000,E1 111.844} C_DIS
LIN {X 0.132,Y -617.756,Z 1009.421,A 0.000,B 0.000,C 90.000,E1 111.844} C_DIS
LIN {X 0.110,Y -610.545,Z 1009.420,A 0.000,B 0.000,C 90.000,E1 111.663} C_DIS
LIN {X 0.263,Y -605.563,Z 1009.419,A 0.000,B 0.000,C 90.000,E1 111.461} C_DIS
LIN {X 0.108,Y -599.880,Z 1009.418,A 0.000,B 0.000,C 90.000,E1 111.227} C_DIS
LIN {X 0.042,Y -593.741,Z 1009.416,A 0.000,B 0.000,C 90.000,E1 110.865} C_DIS
LIN {X -0.211,Y -588.092,Z 1009.414,A 0.000,B 0.000,C 90.000,E1 110.482} C_DIS
LIN {X -0.126,Y -577.105,Z 1009.409,A 0.000,B 0.000,C 90.000,E1 109.577} C_DIS
LIN {X 0.078,Y -572.714,Z 1009.407,A 0.000,B 0.000,C 90.000,E1 109.214} C_DIS
LIN {X 0.217,Y -571.073,Z 1009.406,A 0.000,B 0.000,C 90.000,E1 109.087} C_DIS
LIN {X 0.014,Y -564.479,Z 1009.404,A 0.000,B 0.000,C 90.000,E1 108.725} C_DIS
LIN {X -0.112,Y -550.170,Z 1009.400,A 0.000,B 0.000,C 90.000,E1 108.000} C_DIS
LIN {X 0.003,Y -548.609,Z 1009.399,A 0.000,B 0.000,C 90.000,E1 107.819} C_DIS
LIN {X -0.039,Y -548.604,Z 1009.399,A 0.000,B 0.000,C 90.000,E1 107.819} C_DIS
LIN {X 0.134,Y -548.234,Z 1009.397,A 0.000,B 0.000,C 90.000,E1 107.511} C_DIS
LIN {X -0.100,Y -548.456,Z 1009.392,A 0.000,B 0.000,C 90.000,E1 106.551} C_DIS
LIN {X -0.096,Y -548.996,Z 1009.386,A 0.000,B 0.000,C 90.000,E1 105.426} C_DIS
LIN {X -0.164,Y -550.041,Z 1009.375,A 0.000,B 0.000,C 90.000,E1 103.467} C_DIS
LIN {X 0.142,Y -553.225,Z 1009.355,A 0.000,B 0.000,C 90.000,E1 99.792} C_DIS
LIN {X 0.247,Y -555.100,Z 1009.345,A 0.000,B 0.000,C 90.000,E1 98.106} C_DIS
LIN {X 0.177,Y -556.575,Z 1009.337,A 0.000,B 0.000,C 90.000,E1 96.720} C_DIS
LIN {X -0.064,Y -557.454,Z 1009.333,A 0.000,B 0.000,C 90.000,E1 95.910} C_DIS
LIN {X -0.157,Y -558.592,Z 1009.325,A 0.000,B 0.000,C 90.000,E1 94.531} C_DIS
LIN {X -0.233,Y -559.459,Z 1009.317,A 0.000,B 0.000,C 90.000,E1 93.151} C_DIS
LIN {X 0.030,Y -559.865,Z 1009.313,A 0.000,B 0.000,C 90.000,E1 92.293} C_DIS
LIN {X 0.135,Y -560.766,Z 1009.302,A 0.000,B 0.000,C 90.000,E1 90.344} C_DIS
LIN {X 0.055,Y -561.416,Z 1009.294,A 0.000,B 0.000,C 90.000,E1 88.969} C_DIS
LIN {X -0.100,Y -561.793,Z 1009.288,A 0.000,B 0.000,C 90.000,E1 87.879} C_DIS
LIN {X -0.147,Y -562.036,Z 1009.281,A 0.000,B 0.000,C 90.000,E1 86.502} C_DIS
LIN {X 0.165,Y -562.393,Z 1009.268,A 0.000,B 0.000,C 90.000,E1 84.261} C_DIS
LIN {X 0.220,Y -562.598,Z 1009.261,A 0.000,B 0.000,C 90.000,E1 82.875} C_DIS
LIN {X -0.121,Y -563.047,Z 1009.251,A 0.000,B 0.000,C 90.000,E1 81.254} C_DIS
LIN {X -0.302,Y -563.693,Z 1009.241,A 0.000,B 0.000,C 90.000,E1 79.342} C_DIS
LIN {X 0.064,Y -564.925,Z 1009.227,A 0.000,B 0.000,C 90.000,E1 76.825} C_DIS
LIN {X 0.021,Y -566.297,Z 1009.215,A 0.000,B 0.000,C 90.000,E1 74.629} C_DIS
LIN {X 0.232,Y -567.548,Z 1009.206,A 0.000,B 0.000,C 90.000,E1 72.960} C_DIS
LIN {X -0.243,Y -568.561,Z 1009.198,A 0.000,B 0.000,C 90.000,E1 71.638} C_DIS
LIN {X 0.170,Y -569.782,Z 1009.189,A 0.000,B 0.000,C 90.000,E1 69.953} C_DIS
LIN {X 0.073,Y -570.948,Z 1009.178,A 0.000,B 0.000,C 90.000,E1 68.050} C_DIS
LIN {X -0.306,Y -571.990,Z 1009.168,A 0.000,B 0.000,C 90.000,E1 66.177} C_DIS
LIN {X -0.259,Y -572.666,Z 1009.158,A 0.000,B 0.000,C 90.000,E1 64.537} C_DIS
LIN {X 0.051,Y -573.286,Z 1009.149,A 0.000,B 0.000,C 90.000,E1 62.871} C_DIS
LIN {X -0.137,Y -573.768,Z 1009.140,A 0.000,B 0.000,C 90.000,E1 61.257} C_DIS
LIN {X 0.118,Y -574.205,Z 1009.133,A 0.000,B 0.000,C 90.000,E1 59.871} C_DIS
LIN {X -0.113,Y -574.537,Z 1009.125,A 0.000,B 0.000,C 90.000,E1 58.535} C_DIS
LIN {X -0.174,Y -574.711,Z 1009.119,A 0.000,B 0.000,C 90.000,E1 57.454} C_DIS
LIN {X -0.092,Y -574.962,Z 1009.112,A 0.000,B 0.000,C 90.000,E1 56.087} C_DIS
LIN {X 0.167,Y -575.067,Z 1009.106,A 0.000,B 0.000,C 90.000,E1 54.975} C_DIS
LIN {X -0.041,Y -575.006,Z 1009.100,A 0.000,B 0.000,C 90.000,E1 53.909} C_DIS
LIN {X -0.248,Y -574.837,Z 1009.094,A 0.000,B 0.000,C 90.000,E1 52.844} C_DIS
LIN {X 0.038,Y -574.314,Z 1009.086,A 0.000,B 0.000,C 90.000,E1 51.457} C_DIS
LIN {X 0.170,Y -573.733,Z 1009.080,A 0.000,B 0.000,C 90.000,E1 50.356} C_DIS
LIN {X -0.148,Y -572.982,Z 1009.074,A 0.000,B 0.000,C 90.000,E1 49.299} C_DIS
LIN {X 0.331,Y -572.051,Z 1009.068,A 0.000,B 0.000,C 90.000,E1 48.162} C_DIS
LIN {X -0.139,Y -571.192,Z 1009.063,A 0.000,B 0.000,C 90.000,E1 47.391} C_DIS
LIN {X 0.186,Y -570.209,Z 1009.059,A 0.000,B 0.000,C 90.000,E1 46.539} C_DIS
LIN {X 0.391,Y -569.455,Z 1009.056,A 0.000,B 0.000,C 90.000,E1 45.972} C_DIS
LIN {X -0.018,Y -567.552,Z 1009.050,A 0.000,B 0.000,C 90.000,E1 44.919} C_DIS
LIN {X 0.347,Y -565.476,Z 1009.044,A 0.000,B 0.000,C 90.000,E1 43.785} C_DIS
LIN {X -0.188,Y -563.681,Z 1009.039,A 0.000,B 0.000,C 90.000,E1 43.014} C_DIS
LIN {X -0.268,Y -560.843,Z 1009.033,A 0.000,B 0.000,C 90.000,E1 41.919} C_DIS
LIN {X -0.138,Y -559.210,Z 1009.030,A 0.000,B 0.000,C 90.000,E1 41.353} C_DIS
LIN {X -0.312,Y -556.562,Z 1009.025,A 0.000,B 0.000,C 90.000,E1 40.539} C_DIS
LIN {X 0.273,Y -553.669,Z 1009.020,A 0.000,B 0.000,C 90.000,E1 39.644} C_DIS
LIN {X 0.045,Y -550.350,Z 1009.016,A 0.000,B 0.000,C 90.000,E1 38.830} C_DIS
LIN {X -0.026,Y -546.107,Z 1009.010,A 0.000,B 0.000,C 90.000,E1 37.855} C_DIS
LIN {X 0.087,Y -542.114,Z 1009.006,A 0.000,B 0.000,C 90.000,E1 36.996} C_DIS
LIN {X -0.010,Y -538.616,Z 1009.002,A 0.000,B 0.000,C 90.000,E1 36.297} C_DIS
LIN {X 0.023,Y -534.258,Z 1008.997,A 0.000,B 0.000,C 90.000,E1 35.438} C_DIS
LIN {X -0.298,Y -529.525,Z 1008.992,A 0.000,B 0.000,C 90.000,E1 34.612} C_DIS
LIN {X 0.065,Y -524.463,Z 1008.987,A 0.000,B 0.000,C 90.000,E1 33.706} C_DIS
LIN {X 0.080,Y -519.053,Z 1008.982,A 0.000,B 0.000,C 90.000,E1 32.832} C_DIS
LIN {X -0.045,Y -515.158,Z 1008.979,A 0.000,B 0.000,C 90.000,E1 32.260} C_DIS
LIN {X -0.041,Y -511.031,Z 1008.976,A 0.000,B 0.000,C 90.000,E1 31.671} C_DIS
LIN {X 0.121,Y -507.755,Z 1008.974,A 0.000,B 0.000,C 90.000,E1 31.209} C_DIS
LIN {X 0.077,Y -503.036,Z 1008.970,A 0.000,B 0.000,C 90.000,E1 30.620} C_DIS
LIN {X 0.253,Y -498.033,Z 1008.967,A 0.000,B 0.000,C 90.000,E1 30.001} C_DIS
LIN {X 0.012,Y -491.473,Z 1008.963,A 0.000,B 0.000,C 90.000,E1 29.283} C_DIS
LIN {X 0.125,Y -484.556,Z 1008.959,A 0.000,B 0.000,C 90.000,E1 28.565} C_DIS
LIN {X -0.006,Y -476.375,Z 1008.954,A 0.000,B 0.000,C 90.000,E1 27.769} C_DIS
LIN {X -0.072,Y -467.597,Z 1008.950,A 0.000,B 0.000,C 90.000,E1 26.950} C_DIS
LIN {X 0.239,Y -458.643,Z 1008.945,A 0.000,B 0.000,C 90.000,E1 26.104} C_DIS
LIN {X 0.095,Y -447.906,Z 1008.940,A 0.000,B 0.000,C 90.000,E1 25.207} C_DIS
LIN {X 0.161,Y -422.477,Z 1008.928,A 0.000,B 0.000,C 90.000,E1 22.950} C_DIS
LIN {X -0.089,Y -408.320,Z 1008.920,A 0.000,B 0.000,C 90.000,E1 21.535} C_DIS
LIN {X -0.158,Y -399.958,Z 1008.914,A 0.000,B 0.000,C 90.000,E1 20.610} C_DIS
LIN {X 0.111,Y -395.987,Z 1008.912,A 0.000,B 0.000,C 90.000,E1 20.066} C_DIS
LIN {X 0.039,Y -393.076,Z 1008.909,A 0.000,B 0.000,C 90.000,E1 19.577} C_DIS
LIN {X -0.186,Y -391.217,Z 1008.906,A 0.000,B 0.000,C 90.000,E1 19.033} C_DIS
LIN {X -0.179,Y -390.736,Z 1008.903,A 0.000,B 0.000,C 90.000,E1 18.544} C_DIS
LIN {X -0.155,Y -390.669,Z 1008.902,A 0.000,B 0.000,C 90.000,E1 18.362} C_DIS
LIN {X -0.127,Y -390.799,Z 1008.899,A 0.000,B 0.000,C 90.000,E1 17.819} C_DIS
LIN {X 0.032,Y -395.041,Z 1008.875,A 0.000,B 0.000,C 90.000,E1 13.536} C_DIS
LIN {X -0.061,Y -402.302,Z 1008.848,A 0.000,B 0.000,C 90.000,E1 8.624} C_DIS
LIN {X -0.194,Y -408.283,Z 1008.831,A 0.000,B 0.000,C 90.000,E1 5.511} C_DIS
LIN {X -0.188,Y -412.021,Z 1008.821,A 0.000,B 0.000,C 90.000,E1 3.784} C_DIS
LIN {X -0.170,Y -415.081,Z 1008.813,A 0.000,B 0.000,C 90.000,E1 2.407} C_DIS
LIN {X -0.135,Y -416.946,Z 1008.810,A 0.000,B 0.000,C 90.000,E1 1.718} C_DIS
LIN {X -0.109,Y -419.071,Z 1008.807,A 0.000,B 0.000,C 90.000,E1 1.203} C_DIS
LIN {X -0.097,Y -419.896,Z 1008.806,A 0.000,B 0.000,C 90.000,E1 1.031} C_DIS
LIN {X 0.153,Y -422.853,Z 1008.803,A 0.000,B 0.000,C 90.000,E1 0.573} C_DIS
LIN {X -0.030,Y -425.482,Z 1008.802,A 0.000,B 0.000,C 90.000,E1 0.344} C_DIS
LIN {X -0.211,Y -427.044,Z 1008.801,A 0.000,B 0.000,C 90.000,E1 0.229} C_DIS
LIN {X 0.000,Y -430.047,Z 1008.800,A 0.000,B 0.000,C 90.000,E1 360.000} C_DIS
LIN {X -0.082,Y -437.099,Z 1008.798,A 0.000,B 0.000,C 90.000,E1 359.599} C_DIS
LIN {X 0.078,Y -443.801,Z 1008.796,A 0.000,B 0.000,C 90.000,E1 359.198} C_DIS
LIN {X 0.182,Y -460.297,Z 1008.790,A 0.000,B 0.000,C 90.000,E1 358.224} C_DIS
LIN {X -0.199,Y -476.871,Z 1008.785,A 0.000,B 0.000,C 90.000,E1 357.306} C_DIS
LIN {X -0.138,Y -486.621,Z 1008.782,A 0.000,B 0.000,C 90.000,E1 356.731} C_DIS
LIN {X -0.234,Y -496.436,Z 1008.779,A 0.000,B 0.000,C 90.000,E1 356.159} C_DIS
LIN {X 0.138,Y -506.063,Z 1008.775,A 0.000,B 0.000,C 90.000,E1 355.527} C_DIS
LIN {X 0.135,Y -512.346,Z 1008.773,A 0.000,B 0.000,C 90.000,E1 355.122} C_DIS
LIN {X -0.130,Y -518.470,Z 1008.771,A 0.000,B 0.000,C 90.000,E1 354.723} C_DIS
LIN {X 0.003,Y -524.519,Z 1008.768,A 0.000,B 0.000,C 90.000,E1 354.261} C_DIS
LIN {X -0.073,Y -531.811,Z 1008.765,A 0.000,B 0.000,C 90.000,E1 353.685} C_DIS
LIN {X 0.138,Y -538.757,Z 1008.762,A 0.000,B 0.000,C 90.000,E1 353.053} C_DIS
LIN {X 0.179,Y -544.192,Z 1008.759,A 0.000,B 0.000,C 90.000,E1 352.534} C_DIS
LIN {X -0.065,Y -550.563,Z 1008.755,A 0.000,B 0.000,C 90.000,E1 351.894} C_DIS
LIN {X 0.188,Y -555.371,Z 1008.752,A 0.000,B 0.000,C 90.000,E1 351.319} C_DIS
LIN {X 0.194,Y -560.874,Z 1008.748,A 0.000,B 0.000,C 90.000,E1 350.622} C_DIS
LIN {X -0.059,Y -564.928,Z 1008.745,A 0.000,B 0.000,C 90.000,E1 350.095} C_DIS
LIN {X 0.035,Y -569.341,Z 1008.741,A 0.000,B 0.000,C 90.000,E1 349.398} C_DIS
LIN {X 0.282,Y -575.726,Z 1008.735,A 0.000,B 0.000,C 90.000,E1 348.285} C_DIS
LIN {X -0.100,Y -579.382,Z 1008.731,A 0.000,B 0.000,C 90.000,E1 347.645} C_DIS
LIN {X -0.093,Y -584.115,Z 1008.726,A 0.000,B 0.000,C 90.000,E1 346.700} C_DIS
LIN {X -0.257,Y -589.192,Z 1008.720,A 0.000,B 0.000,C 90.000,E1 345.644} C_DIS
LIN {X 0.172,Y -592.249,Z 1008.716,A 0.000,B 0.000,C 90.000,E1 344.936} C_DIS
LIN {X -0.316,Y -596.875,Z 1008.711,A 0.000,B 0.000,C 90.000,E1 343.921} C_DIS
LIN {X 0.009,Y -603.383,Z 1008.702,A 0.000,B 0.000,C 90.000,E1 342.308} C_DIS
LIN {X 0.152,Y -608.373,Z 1008.695,A 0.000,B 0.000,C 90.000,E1 340.986} C_DIS
LIN {X 0.268,Y -612.155,Z 1008.689,A 0.000,B 0.000,C 90.000,E1 339.934} C_DIS
LIN {X -0.304,Y -614.617,Z 1008.684,A 0.000,B 0.000,C 90.000,E1 339.209} C_DIS
LIN {X -0.091,Y -617.801,Z 1008.679,A 0.000,B 0.000,C 90.000,E1 338.156} C_DIS
LIN {X -0.091,Y -622.261,Z 1008.670,A 0.000,B 0.000,C 90.000,E1 336.613} C_DIS
LIN {X -0.095,Y -624.266,Z 1008.666,A 0.000,B 0.000,C 90.000,E1 335.845} C_DIS
LIN {X 0.247,Y -626.785,Z 1008.660,A 0.000,B 0.000,C 90.000,E1 334.793} C_DIS
LIN {X 0.341,Y -629.693,Z 1008.653,A 0.000,B 0.000,C 90.000,E1 333.512} C_DIS
LIN {X -0.168,Y -630.739,Z 1008.650,A 0.000,B 0.000,C 90.000,E1 333.050} C_DIS
LIN {X -0.007,Y -633.124,Z 1008.643,A 0.000,B 0.000,C 90.000,E1 331.769} C_DIS
LIN {X -0.020,Y -635.708,Z 1008.635,A 0.000,B 0.000,C 90.000,E1 330.255} C_DIS
LIN {X 0.104,Y -636.887,Z 1008.631,A 0.000,B 0.000,C 90.000,E1 329.488} C_DIS
LIN {X 0.055,Y -638.259,Z 1008.625,A 0.000,B 0.000,C 90.000,E1 328.486} C_DIS
LIN {X -0.134,Y -639.810,Z 1008.618,A 0.000,B 0.000,C 90.000,E1 327.248} C_DIS
LIN {X -0.287,Y -641.163,Z 1008.611,A 0.000,B 0.000,C 90.000,E1 326.008} C_DIS
LIN {X 0.067,Y -641.945,Z 1008.606,A 0.000,B 0.000,C 90.000,E1 324.975} C_DIS
LIN {X -0.097,Y -642.561,Z 1008.600,A 0.000,B 0.000,C 90.000,E1 323.989} C_DIS
LIN {X 0.052,Y -643.177,Z 1008.592,A 0.000,B 0.000,C 90.000,E1 322.477} C_DIS
LIN {X 0.123,Y -643.718,Z 1008.582,A 0.000,B 0.000,C 90.000,E1 320.723} C_DIS
LIN {X -0.046,Y -644.727,Z 1008.568,A 0.000,B 0.000,C 90.000,E1 318.243} C_DIS
LIN {X 0.072,Y -645.376,Z 1008.561,A 0.000,B 0.000,C 90.000,E1 316.986} C_DIS
LIN {X 0.135,Y -646.155,Z 1008.553,A 0.000,B 0.000,C 90.000,E1 315.486} C_DIS
LIN {X 0.093,Y -647.393,Z 1008.542,A 0.000,B 0.000,C 90.000,E1 313.500} C_DIS
LIN {X 0.199,Y -648.306,Z 1008.534,A 0.000,B 0.000,C 90.000,E1 312.000} C_DIS
LIN {X -0.121,Y -649.078,Z 1008.525,A 0.000,B 0.000,C 90.000,E1 310.539} C_DIS
LIN {X 0.059,Y -649.673,Z 1008.517,A 0.000,B 0.000,C 90.000,E1 309.036} C_DIS
LIN {X -0.166,Y -650.236,Z 1008.509,A 0.000,B 0.000,C 90.000,E1 307.569} C_DIS
LIN {X 0.213,Y -650.554,Z 1008.502,A 0.000,B 0.000,C 90.000,E1 306.297} C_DIS
LIN {X 0.160,Y -650.726,Z 1008.496,A 0.000,B 0.000,C 90.000,E1 305.311} C_DIS
LIN {X 0.133,Y -651.268,Z 1008.484,A 0.000,B 0.000,C 90.000,E1 303.086} C_DIS
LIN {X -0.009,Y -654.530,Z 1008.461,A 0.000,B 0.000,C 90.000,E1 298.899} C_DIS
LIN {X 0.170,Y -657.293,Z 1008.448,A 0.000,B 0.000,C 90.000,E1 296.668} C_DIS
LIN {X -0.101,Y -658.909,Z 1008.441,A 0.000,B 0.000,C 90.000,E1 295.463} C_DIS
LIN {X 0.000,Y -659.774,Z 1008.437,A 0.000,B 0.000,C 90.000,E1 294.719} C_DIS
LIN {X 0.384,Y -660.477,Z 1008.433,A 0.000,B 0.000,C 90.000,E1 293.951} C_DIS
LIN {X -0.101,Y -660.933,Z 1008.429,A 0.000,B 0.000,C 90.000,E1 293.259} C_DIS
LIN {X -0.103,Y -661.169,Z 1008.427,A 0.000,B 0.000,C 90.000,E1 292.770} C_DIS
LIN {X 0.026,Y -661.230,Z 1008.422,A 0.000,B 0.000,C 90.000,E1 292.025} C_DIS
LIN {X 0.031,Y -660.860,Z 1008.420,A 0.000,B 0.000,C 90.000,E1 291.535} C_DIS
LIN {X 0.036,Y -659.855,Z 1008.417,A 0.000,B 0.000,C 90.000,E1 291.046} C_DIS
LIN {X 0.154,Y -659.178,Z 1008.416,A 0.000,B 0.000,C 90.000,E1 290.791} C_DIS
LIN {X 0.035,Y -657.626,Z 1008.414,A 0.000,B 0.000,C 90.000,E1 290.556} C_DIS
LIN {X -0.311,Y -656.151,Z 1008.413,A 0.000,B 0.000,C 90.000,E1 290.301} C_DIS
LIN {X -0.259,Y -655.302,Z 1008.412,A 0.000,B 0.000,C 90.000,E1 290.174} C_DIS
LIN {X 0.404,Y -654.018,Z 1008.411,A 0.000,B 0.000,C 90.000,E1 289.993} C_DIS
LIN {X 0.230,Y -652.168,Z 1008.411,A 0.000,B 0.000,C 90.000,E1 289.885} C_DIS
LIN {X -0.304,Y -648.249,Z 1008.409,A 0.000,B 0.000,C 90.000,E1 289.631} C_DIS
LIN {X -0.020,Y -640.347,Z 1008.406,A 0.000,B 0.000,C 90.000,E1 289.141} C_DIS
LIN {X -0.092,Y -634.254,Z 1008.405,A 0.000,B 0.000,C 90.000,E1 288.852} C_DIS
LIN {X -0.169,Y -631.317,Z 1008.404,A 0.000,B 0.000,C 90.000,E1 288.652} C_DIS
LIN {X -0.207,Y -631.277,Z 1008.404,A 0.000,B 0.000,C 90.000,E1 288.652} C_DIS
LIN {X -0.128,Y -630.820,Z 1008.403,A 0.000,B 0.000,C 90.000,E1 288.489} C_DIS
LIN {X -0.172,Y -630.814,Z 1008.403,A 0.000,B 0.000,C 90.000,E1 288.489} C_DIS
LIN {X -0.268,Y -633.219,Z 1008.400,A 0.000,B 0.000,C 90.000,E1 288.055} C_DIS
LIN {X 0.237,Y -640.434,Z 1008.394,A 0.000,B 0.000,C 90.000,E1 286.913} C_DIS
LIN {X -0.195,Y -644.745,Z 1008.390,A 0.000,B 0.000,C 90.000,E1 286.205} C_DIS
LIN {X 0.146,Y -647.855,Z 1008.387,A 0.000,B 0.000,C 90.000,E1 285.552} C_DIS
LIN {X 0.008,Y -648.909,Z 1008.385,A 0.000,B 0.000,C 90.000,E1 285.315} C_DIS
LIN {X -0.096,Y -650.670,Z 1008.382,A 0.000,B 0.000,C 90.000,E1 284.828} C_DIS
LIN {X -0.228,Y -651.446,Z 1008.381,A 0.000,B 0.000,C 90.000,E1 284.592} C_DIS
LIN {X 0.148,Y -652.709,Z 1008.378,A 0.000,B 0.000,C 90.000,E1 284.064} C_DIS
LIN {X -0.219,Y -654.035,Z 1008.374,A 0.000,B 0.000,C 90.000,E1 283.355} C_DIS
LIN {X 0.061,Y -654.685,Z 1008.370,A 0.000,B 0.000,C 90.000,E1 282.591} C_DIS
LIN {X -0.056,Y -654.868,Z 1008.369,A 0.000,B 0.000,C 90.000,E1 282.355} C_DIS
LIN {X 0.230,Y -654.894,Z 1008.365,A 0.000,B 0.000,C 90.000,E1 281.591} C_DIS
LIN {X -0.136,Y -654.627,Z 1008.362,A 0.000,B 0.000,C 90.000,E1 281.130} C_DIS
LIN {X 0.267,Y -654.090,Z 1008.359,A 0.000,B 0.000,C 90.000,E1 280.602} C_DIS
LIN {X -0.095,Y -653.258,Z 1008.356,A 0.000,B 0.000,C 90.000,E1 280.141} C_DIS
LIN {X 0.164,Y -651.507,Z 1008.352,A 0.000,B 0.000,C 90.000,E1 279.378} C_DIS
LIN {X -0.209,Y -649.918,Z 1008.349,A 0.000,B 0.000,C 90.000,E1 278.916} C_DIS
LIN {X 0.053,Y -647.918,Z 1008.347,A 0.000,B 0.000,C 90.000,E1 278.398} C_DIS
LIN {X 0.271,Y -644.886,Z 1008.343,A 0.000,B 0.000,C 90.000,E1 277.757} C_DIS
LIN {X -0.140,Y -641.648,Z 1008.341,A 0.000,B 0.000,C 90.000,E1 277.296} C_DIS
LIN {X -0.062,Y -636.860,Z 1008.337,A 0.000,B 0.000,C 90.000,E1 276.663} C_DIS
LIN {X 0.111,Y -632.255,Z 1008.334,A 0.000,B 0.000,C 90.000,E1 276.144} C_DIS
LIN {X -0.324,Y -626.103,Z 1008.331,A 0.000,B 0.000,C 90.000,E1 275.568} C_DIS
LIN {X 0.181,Y -619.454,Z 1008.328,A 0.000,B 0.000,C 90.000,E1 274.935} C_DIS
LIN {X -0.252,Y -613.598,Z 1008.325,A 0.000,B 0.000,C 90.000,E1 274.531} C_DIS
LIN {X -0.186,Y -605.835,Z 1008.322,A 0.000,B 0.000,C 90.000,E1 274.012} C_DIS
LIN {X 0.146,Y -599.288,Z 1008.320,A 0.000,B 0.000,C 90.000,E1 273.612} C_DIS
LIN {X 0.236,Y -592.359,Z 1008.318,A 0.000,B 0.000,C 90.000,E1 273.269} C_DIS
LIN {X -0.246,Y -585.032,Z 1008.317,A 0.000,B 0.000,C 90.000,E1 273.037} C_DIS
LIN {X -0.164,Y -577.395,Z 1008.316,A 0.000,B 0.000,C 90.000,E1 272.808} C_DIS
LIN {X 0.218,Y -571.698,Z 1008.315,A 0.000,B 0.000,C 90.000,E1 272.636} C_DIS
LIN {X 0.196,Y -565.077,Z 1008.314,A 0.000,B 0.000,C 90.000,E1 272.522} C_DIS
LIN {X 0.277,Y -558.134,Z 1008.314,A 0.000,B 0.000,C 90.000,E1 272.465} C_DIS
LIN {X 0.231,Y -543.875,Z 1008.314,A 0.000,B 0.000,C 90.000,E1 272.465} C_DIS
LIN {X 0.144,Y -542.747,Z 1008.312,A 0.000,B 0.000,C 90.000,E1 272.178} C_DIS
LIN {X 0.220,Y -542.129,Z 1008.309,A 0.000,B 0.000,C 90.000,E1 271.604} C_DIS
LIN {X -0.168,Y -541.009,Z 1008.300,A 0.000,B 0.000,C 90.000,E1 269.943} C_DIS
LIN {X -0.058,Y -540.111,Z 1008.292,A 0.000,B 0.000,C 90.000,E1 268.511} C_DIS
LIN {X 0.015,Y -539.544,Z 1008.287,A 0.000,B 0.000,C 90.000,E1 267.650} C_DIS
LIN {X 0.162,Y -537.997,Z 1008.276,A 0.000,B 0.000,C 90.000,E1 265.641} C_DIS
LIN {X -0.230,Y -536.399,Z 1008.265,A 0.000,B 0.000,C 90.000,E1 263.685} C_DIS
LIN {X -0.107,Y -535.127,Z 1008.257,A 0.000,B 0.000,C 90.000,E1 262.243} C_DIS
LIN {X 0.066,Y -533.717,Z 1008.249,A 0.000,B 0.000,C 90.000,E1 260.792} C_DIS
LIN {X 0.167,Y -532.450,Z 1008.243,A 0.000,B 0.000,C 90.000,E1 259.634} C_DIS
LIN {X -0.061,Y -530.262,Z 1008.231,A 0.000,B 0.000,C 90.000,E1 257.645} C_DIS
LIN {X 0.230,Y -528.744,Z 1008.223,A 0.000,B 0.000,C 90.000,E1 256.172} C_DIS
LIN {X 0.137,Y -526.780,Z 1008.214,A 0.000,B 0.000,C 90.000,E1 254.448} C_DIS
LIN {X 0.001,Y -524.900,Z 1008.204,A 0.000,B 0.000,C 90.000,E1 252.725} C_DIS
LIN {X -0.025,Y -523.273,Z 1008.196,A 0.000,B 0.000,C 90.000,E1 251.275} C_DIS
LIN {X -0.059,Y -521.786,Z 1008.190,A 0.000,B 0.000,C 90.000,E1 250.115} C_DIS
LIN {X -0.195,Y -518.810,Z 1008.177,A 0.000,B 0.000,C 90.000,E1 247.794} C_DIS
LIN {X -0.108,Y -517.208,Z 1008.170,A 0.000,B 0.000,C 90.000,E1 246.613} C_DIS
LIN {X 0.294,Y -515.071,Z 1008.162,A 0.000,B 0.000,C 90.000,E1 245.101} C_DIS
LIN {X 0.076,Y -513.302,Z 1008.155,A 0.000,B 0.000,C 90.000,E1 243.948} C_DIS
LIN {X -0.061,Y -510.917,Z 1008.147,A 0.000,B 0.000,C 90.000,E1 242.487} C_DIS
LIN {X -0.016,Y -508.568,Z 1008.139,A 0.000,B 0.000,C 90.000,E1 241.001} C_DIS
LIN {X -0.213,Y -505.989,Z 1008.131,A 0.000,B 0.000,C 90.000,E1 239.537} C_DIS
LIN {X -0.071,Y -503.755,Z 1008.124,A 0.000,B 0.000,C 90.000,E1 238.329} C_DIS
LIN {X -0.087,Y -500.802,Z 1008.116,A 0.000,B 0.000,C 90.000,E1 236.834} C_DIS
LIN {X 0.258,Y -496.156,Z 1008.104,A 0.000,B 0.000,C 90.000,E1 234.689} C_DIS
LIN {X -0.185,Y -491.725,Z 1008.094,A 0.000,B 0.000,C 90.000,E1 232.924} C_DIS
LIN {X -0.131,Y -487.288,Z 1008.084,A 0.000,B 0.000,C 90.000,E1 231.090} C_DIS
LIN {X 0.137,Y -483.017,Z 1008.074,A 0.000,B 0.000,C 90.000,E1 229.218} C_DIS
LIN {X 0.183,Y -475.536,Z 1008.055,A 0.000,B 0.000,C 90.000,E1 225.810} C_DIS
LIN {X 0.120,Y -471.747,Z 1008.044,A 0.000,B 0.000,C 90.000,E1 223.947} C_DIS
LIN {X -0.013,Y -467.774,Z 1008.034,A 0.000,B 0.000,C 90.000,E1 222.081} C_DIS
LIN {X 0.056,Y -464.355,Z 1008.025,A 0.000,B 0.000,C 90.000,E1 220.496} C_DIS
LIN {X 0.058,Y -460.759,Z 1008.016,A 0.000,B 0.000,C 90.000,E1 218.910} C_DIS
LIN {X 0.067,Y -456.553,Z 1008.006,A 0.000,B 0.000,C 90.000,E1 216.996} C_DIS
LIN {X -0.203,Y -452.302,Z 1007.995,A 0.000,B 0.000,C 90.000,E1 215.105} C_DIS
LIN {X 0.104,Y -448.719,Z 1007.986,A 0.000,B 0.000,C 90.000,E1 213.452} C_DIS
LIN {X 0.030,Y -445.954,Z 1007.979,A 0.000,B 0.000,C 90.000,E1 212.163} C_DIS
LIN {X 0.078,Y -440.995,Z 1007.966,A 0.000,B 0.000,C 90.000,E1 209.873} C_DIS
LIN {X 0.000,Y -438.770,Z 1007.961,A 0.000,B 0.000,C 90.000,E1 208.899} C_DIS
LIN {X -0.031,Y -434.297,Z 1007.950,A 0.000,B 0.000,C 90.000,E1 206.924} C_DIS
LIN {X 0.015,Y -429.047,Z 1007.937,A 0.000,B 0.000,C 90.000,E1 204.591} C_DIS
LIN {X 0.161,Y -425.273,Z 1007.927,A 0.000,B 0.000,C 90.000,E1 202.898} C_DIS
LIN {X -0.252,Y -418.133,Z 1007.909,A 0.000,B 0.000,C 90.000,E1 199.577} C_DIS
LIN {X -0.097,Y -414.230,Z 1007.897,A 0.000,B 0.000,C 90.000,E1 197.511} C_DIS
LIN {X 0.106,Y -410.661,Z 1007.886,A 0.000,B 0.000,C 90.000,E1 195.426} C_DIS
LIN {X -0.163,Y -406.304,Z 1007.870,A 0.000,B 0.000,C 90.000,E1 192.703} C_DIS
LIN {X -0.039,Y -402.451,Z 1007.855,A 0.000,B 0.000,C 90.000,E1 189.905} C_DIS
LIN {X -0.047,Y -401.430,Z 1007.849,A 0.000,B 0.000,C 90.000,E1 188.859} C_DIS
LIN {X -0.072,Y -401.373,Z 1007.843,A 0.000,B 0.000,C 90.000,E1 187.814} C_DIS
LIN {X -0.082,Y -401.557,Z 1007.841,A 0.000,B 0.000,C 90.000,E1 187.466} C_DIS
LIN {X -0.142,Y -402.011,Z 1007.840,A 0.000,B 0.000,C 90.000,E1 187.125} C_DIS
LIN {X -0.186,Y -403.858,Z 1007.835,A 0.000,B 0.000,C 90.000,E1 186.258} C_DIS
LIN {X -0.211,Y -404.391,Z 1007.834,A 0.000,B 0.000,C 90.000,E1 186.087} C_DIS
LIN {X 0.083,Y -406.552,Z 1007.831,A 0.000,B 0.000,C 90.000,E1 185.511} C_DIS
LIN {X 0.087,Y -408.315,Z 1007.829,A 0.000,B 0.000,C 90.000,E1 185.163} C_DIS
LIN {X -0.035,Y -411.151,Z 1007.826,A 0.000,B 0.000,C 90.000,E1 184.702} C_DIS
LIN {X 0.028,Y -413.550,Z 1007.824,A 0.000,B 0.000,C 90.000,E1 184.359} C_DIS
LIN {X 0.062,Y -425.963,Z 1007.816,A 0.000,B 0.000,C 90.000,E1 182.865} C_DIS
LIN {X -0.111,Y -434.432,Z 1007.811,A 0.000,B 0.000,C 90.000,E1 181.949} C_DIS
LIN {X 0.158,Y -444.089,Z 1007.805,A 0.000,B 0.000,C 90.000,E1 180.802} C_DIS
LIN {X 0.082,Y -453.596,Z 1007.799,A 0.000,B 0.000,C 90.000,E1 179.714} C_DIS
LIN {X 0.011,Y -461.582,Z 1007.793,A 0.000,B 0.000,C 90.000,E1 178.797} C_DIS
LIN {X -0.179,Y -469.421,Z 1007.788,A 0.000,B 0.000,C 90.000,E1 177.879} C_DIS
LIN {X -0.100,Y -479.570,Z 1007.781,A 0.000,B 0.000,C 90.000,E1 176.617} C_DIS
LIN {X -0.019,Y -484.340,Z 1007.778,A 0.000,B 0.000,C 90.000,E1 175.988} C_DIS
LIN {X -0.007,Y -494.299,Z 1007.770,A 0.000,B 0.000,C 90.000,E1 174.609} C_DIS
LIN {X 0.046,Y -502.611,Z 1007.763,A 0.000,B 0.000,C 90.000,E1 173.394} C_DIS
LIN {X -0.076,Y -511.459,Z 1007.756,A 0.000,B 0.000,C 90.000,E1 172.064} C_DIS
LIN {X 0.246,Y -518.845,Z 1007.749,A 0.000,B 0.000,C 90.000,E1 170.849} C_DIS
LIN {X -0.094,Y -530.128,Z 1007.739,A 0.000,B 0.000,C 90.000,E1 168.993} C_DIS
LIN {X -0.089,Y -537.792,Z 1007.732,A 0.000,B 0.000,C 90.000,E1 167.701} C_DIS
LIN {X 0.029,Y -545.166,Z 1007.725,A 0.000,B 0.000,C 90.000,E1 166.408} C_DIS
LIN {X 0.015,Y -551.593,Z 1007.718,A 0.000,B 0.000,C 90.000,E1 165.283} C_DIS
LIN {X 0.093,Y -557.821,Z 1007.712,A 0.000,B 0.000,C 90.000,E1 164.157} C_DIS
LIN {X 0.110,Y -562.332,Z 1007.707,A 0.000,B 0.000,C 90.000,E1 163.323} C_DIS
LIN {X -0.320,Y -568.751,Z 1007.701,A 0.000,B 0.000,C 90.000,E1 162.127} C_DIS
LIN {X 0.063,Y -574.986,Z 1007.694,A 0.000,B 0.000,C 90.000,E1 160.859} C_DIS
LIN {X 0.001,Y -580.817,Z 1007.687,A 0.000,B 0.000,C 90.000,E1 159.645} C_DIS
LIN {X -0.244,Y -585.738,Z 1007.681,A 0.000,B 0.000,C 90.000,E1 158.592} C_DIS
LIN {X 0.122,Y -590.321,Z 1007.675,A 0.000,B 0.000,C 90.000,E1 157.486} C_DIS
LIN {X 0.000,Y -594.596,Z 1007.669,A 0.000,B 0.000,C 90.000,E1 156.433} C_DIS
LIN {X -0.192,Y -596.619,Z 1007.666,A 0.000,B 0.000,C 90.000,E1 155.921} C_DIS
LIN {X 0.016,Y -600.299,Z 1007.660,A 0.000,B 0.000,C 90.000,E1 154.845} C_DIS
LIN {X 0.278,Y -603.674,Z 1007.654,A 0.000,B 0.000,C 90.000,E1 153.768} C_DIS
LIN {X 0.042,Y -606.799,Z 1007.649,A 0.000,B 0.000,C 90.000,E1 152.743} C_DIS
LIN {X 0.046,Y -611.284,Z 1007.640,A 0.000,B 0.000,C 90.000,E1 151.179} C_DIS
LIN {X 0.201,Y -614.139,Z 1007.634,A 0.000,B 0.000,C 90.000,E1 150.127} C_DIS
LIN {X -0.164,Y -617.656,Z 1007.627,A 0.000,B 0.000,C 90.000,E1 148.869} C_DIS
LIN {X -0.173,Y -621.750,Z 1007.618,A 0.000,B 0.000,C 90.000,E1 147.327} C_DIS
LIN {X 0.055,Y -626.486,Z 1007.609,A 0.000,B 0.000,C 90.000,E1 145.515} C_DIS
LIN {X -0.106,Y -631.222,Z 1007.599,A 0.000,B 0.000,C 90.000,E1 143.749} C_DIS
LIN {X 0.345,Y -635.169,Z 1007.590,A 0.000,B 0.000,C 90.000,E1 142.190} C_DIS
LIN {X -0.029,Y -638.470,Z 1007.583,A 0.000,B 0.000,C 90.000,E1 140.964} C_DIS
LIN {X 0.045,Y -641.674,Z 1007.576,A 0.000,B 0.000,C 90.000,E1 139.703} C_DIS
LIN {X 0.188,Y -644.212,Z 1007.571,A 0.000,B 0.000,C 90.000,E1 138.690} C_DIS
LIN {X -0.128,Y -647.382,Z 1007.564,A 0.000,B 0.000,C 90.000,E1 137.472} C_DIS
LIN {X -0.158,Y -653.477,Z 1007.551,A 0.000,B 0.000,C 90.000,E1 135.243} C_DIS
LIN {X -0.018,Y -661.086,Z 1007.538,A 0.000,B 0.000,C 90.000,E1 132.771} C_DIS
LIN {X -0.069,Y -665.889,Z 1007.530,A 0.000,B 0.000,C 90.000,E1 131.310} C_DIS
LIN {X -0.034,Y -670.567,Z 1007.521,A 0.000,B 0.000,C 90.000,E1 129.850} C_DIS
LIN {X -0.364,Y -673.478,Z 1007.516,A 0.000,B 0.000,C 90.000,E1 128.910} C_DIS
LIN {X -0.108,Y -676.940,Z 1007.509,A 0.000,B 0.000,C 90.000,E1 127.684} C_DIS
LIN {X 0.211,Y -680.342,Z 1007.503,A 0.000,B 0.000,C 90.000,E1 126.457} C_DIS
LIN {X 0.195,Y -684.235,Z 1007.495,A 0.000,B 0.000,C 90.000,E1 125.025} C_DIS
LIN {X -0.166,Y -687.426,Z 1007.488,A 0.000,B 0.000,C 90.000,E1 123.865} C_DIS
LIN {X -0.318,Y -689.263,Z 1007.484,A 0.000,B 0.000,C 90.000,E1 123.166} C_DIS
LIN {X -0.132,Y -694.063,Z 1007.474,A 0.000,B 0.000,C 90.000,E1 121.258} C_DIS
LIN {X -0.357,Y -696.300,Z 1007.468,A 0.000,B 0.000,C 90.000,E1 120.335} C_DIS
LIN {X -0.199,Y -697.742,Z 1007.464,A 0.000,B 0.000,C 90.000,E1 119.617} C_DIS
LIN {X -0.372,Y -699.308,Z 1007.459,A 0.000,B 0.000,C 90.000,E1 118.693} C_DIS
LIN {X 0.087,Y -700.545,Z 1007.454,A 0.000,B 0.000,C 90.000,E1 117.719} C_DIS
LIN {X 0.096,Y -702.018,Z 1007.444,A 0.000,B 0.000,C 90.000,E1 115.848} C_DIS
LIN {X 0.273,Y -702.693,Z 1007.438,A 0.000,B 0.000,C 90.000,E1 114.899} C_DIS
LIN {X 0.180,Y -702.872,Z 1007.435,A 0.000,B 0.000,C 90.000,E1 114.207} C_DIS
LIN {X -0.191,Y -702.253,Z 1007.432,A 0.000,B 0.000,C 90.000,E1 113.770} C_DIS
LIN {X 0.086,Y -701.862,Z 1007.431,A 0.000,B 0.000,C 90.000,E1 113.515} C_DIS
LIN {X -0.289,Y -699.896,Z 1007.428,A 0.000,B 0.000,C 90.000,E1 113.078} C_DIS
LIN {X -0.021,Y -698.697,Z 1007.427,A 0.000,B 0.000,C 90.000,E1 112.823} C_DIS
LIN {X 0.109,Y -697.689,Z 1007.426,A 0.000,B 0.000,C 90.000,E1 112.695} C_DIS
LIN {X -0.028,Y -696.186,Z 1007.426,A 0.000,B 0.000,C 90.000,E1 112.589} C_DIS
LIN {X -0.224,Y -690.131,Z 1007.423,A 0.000,B 0.000,C 90.000,E1 112.206} C_DIS
LIN {X 0.203,Y -687.780,Z 1007.423,A 0.000,B 0.000,C 90.000,E1 112.078} C_DIS
LIN {X -0.267,Y -685.010,Z 1007.422,A 0.000,B 0.000,C 90.000,E1 112.025} C_DIS
LIN {X -0.057,Y -682.067,Z 1007.422,A 0.000,B 0.000,C 90.000,E1 111.950} C_DIS
LIN {X 0.098,Y -674.958,Z 1007.421,A 0.000,B 0.000,C 90.000,E1 111.844} C_DIS
LIN {X 0.043,Y -618.206,Z 1007.421,A 0.000,B 0.000,C 90.000,E1 111.844} C_DIS
LIN {X 0.051,Y -610.856,Z 1007.420,A 0.000,B 0.000,C 90.000,E1 111.663} C_DIS
LIN {X 0.169,Y -604.423,Z 1007.419,A 0.000,B 0.000,C 90.000,E1 111.408} C_DIS
LIN {X 0.068,Y -600.115,Z 1007.418,A 0.000,B 0.000,C 90.000,E1 111.227} C_DIS
LIN {X -0.274,Y -594.321,Z 1007.416,A 0.000,B 0.000,C 90.000,E1 110.918} C_DIS
LIN {X 0.066,Y -587.332,Z 1007.413,A 0.000,B 0.000,C 90.000,E1 110.375} C_DIS
LIN {X 0.005,Y -577.487,Z 1007.409,A 0.000,B 0.000,C 90.000,E1 109.577} C_DIS
LIN {X -0.192,Y -571.566,Z 1007.406,A 0.000,B 0.000,C 90.000,E1 109.141} C_DIS
LIN {X -0.138,Y -563.129,Z 1007.404,A 0.000,B 0.000,C 90.000,E1 108.652} C_DIS
LIN {X -0.294,Y -550.060,Z 1007.400,A 0.000,B 0.000,C 90.000,E1 108.000} C_DIS
LIN {X -0.093,Y -548.677,Z 1007.399,A 0.000,B 0.000,C 90.000,E1 107.819} C_DIS
LIN {X -0.134,Y -548.657,Z 1007.399,A 0.000,B 0.000,C 90.000,E1 107.819} C_DIS
LIN {X 0.164,Y -548.291,Z 1007.397,A 0.000,B 0.000,C 90.000,E1 107.511} C_DIS
LIN {X -0.063,Y -549.055,Z 1007.386,A 0.000,B 0.000,C 90.000,E1 105.426} C_DIS
LIN {X -0.130,Y -550.098,Z 1007.375,A 0.000,B 0.000,C 90.000,E1 103.467} C_DIS
LIN {X -0.247,Y -553.553,Z 1007.353,A 0.000,B 0.000,C 90.000,E1 99.557} C_DIS
LIN {X -0.266,Y -555.126,Z 1007.345,A 0.000,B 0.000,C 90.000,E1 98.163} C_DIS
LIN {X 0.214,Y -556.603,Z 1007.338,A 0.000,B 0.000,C 90.000,E1 96.720} C_DIS
LIN {X 0.042,Y -557.699,Z 1007.331,A 0.000,B 0.000,C 90.000,E1 95.625} C_DIS
LIN {X -0.040,Y -558.765,Z 1007.324,A 0.000,B 0.000,C 90.000,E1 94.245} C_DIS
LIN {X -0.110,Y -559.613,Z 1007.316,A 0.000,B 0.000,C 90.000,E1 92.865} C_DIS
LIN {X -0.016,Y -560.481,Z 1007.305,A 0.000,B 0.000,C 90.000,E1 90.917} C_DIS
LIN {X -0.101,Y -561.195,Z 1007.297,A 0.000,B 0.000,C 90.000,E1 89.542} C_DIS
LIN {X -0.161,Y -561.768,Z 1007.290,A 0.000,B 0.000,C 90.000,E1 88.165} C_DIS
LIN {X -0.205,Y -562.002,Z 1007.282,A 0.000,B 0.000,C 90.000,E1 86.788} C_DIS
LIN {X 0.205,Y -562.393,Z 1007.268,A 0.000,B 0.000,C 90.000,E1 84.261} C_DIS
LIN {X -0.067,Y -562.705,Z 1007.258,A 0.000,B 0.000,C 90.000,E1 82.356} C_DIS
LIN {X -0.083,Y -563.047,Z 1007.251,A 0.000,B 0.000,C 90.000,E1 81.254} C_DIS
LIN {X -0.263,Y -563.692,Z 1007.241,A 0.000,B 0.000,C 90.000,E1 79.342} C_DIS
LIN {X -0.062,Y -564.734,Z 1007.228,A 0.000,B 0.000,C 90.000,E1 77.117} C_DIS
LIN {X 0.128,Y -565.937,Z 1007.218,A 0.000,B 0.000,C 90.000,E1 75.172} C_DIS
LIN {X -0.112,Y -567.760,Z 1007.204,A 0.000,B 0.000,C 90.000,E1 72.725} C_DIS
LIN {X 0.133,Y -568.741,Z 1007.196,A 0.000,B 0.000,C 90.000,E1 71.329} C_DIS
LIN {X -0.329,Y -569.760,Z 1007.189,A 0.000,B 0.000,C 90.000,E1 70.007} C_DIS
LIN {X 0.109,Y -570.901,Z 1007.178,A 0.000,B 0.000,C 90.000,E1 68.050} C_DIS
LIN {X 0.295,Y -571.606,Z 1007.171,A 0.000,B 0.000,C 90.000,E1 66.666} C_DIS
LIN {X 0.082,Y -572.021,Z 1007.166,A 0.000,B 0.000,C 90.000,E1 65.869} C_DIS
LIN {X 0.126,Y -572.700,Z 1007.157,A 0.000,B 0.000,C 90.000,E1 64.229} C_DIS
LIN {X -0.077,Y -573.245,Z 1007.148,A 0.000,B 0.000,C 90.000,E1 62.615} C_DIS
LIN {X -0.107,Y -573.671,Z 1007.140,A 0.000,B 0.000,C 90.000,E1 61.257} C_DIS
LIN {X 0.146,Y -574.110,Z 1007.133,A 0.000,B 0.000,C 90.000,E1 59.871} C_DIS
LIN {X 0.049,Y -574.467,Z 1007.124,A 0.000,B 0.000,C 90.000,E1 58.250} C_DIS
LIN {X 0.105,Y -574.761,Z 1007.113,A 0.000,B 0.000,C 90.000,E1 56.342} C_DIS
LIN {X 0.041,Y -574.904,Z 1007.107,A 0.000,B 0.000,C 90.000,E1 55.261} C_DIS
LIN {X -0.171,Y -574.869,Z 1007.101,A 0.000,B 0.000,C 90.000,E1 54.196} C_DIS
LIN {X 0.079,Y -574.699,Z 1007.095,A 0.000,B 0.000,C 90.000,E1 53.084} C_DIS
LIN {X -0.084,Y -574.570,Z 1007.092,A 0.000,B 0.000,C 90.000,E1 52.557} C_DIS
LIN {X 0.051,Y -574.126,Z 1007.086,A 0.000,B 0.000,C 90.000,E1 51.457} C_DIS
LIN {X 0.181,Y -573.526,Z 1007.080,A 0.000,B 0.000,C 90.000,E1 50.356} C_DIS
LIN {X -0.007,Y -572.536,Z 1007.072,A 0.000,B 0.000,C 90.000,E1 49.013} C_DIS
LIN {X 0.334,Y -571.821,Z 1007.068,A 0.000,B 0.000,C 90.000,E1 48.162} C_DIS
LIN {X -0.137,Y -570.954,Z 1007.063,A 0.000,B 0.000,C 90.000,E1 47.391} C_DIS
LIN {X 0.186,Y -569.932,Z 1007.059,A 0.000,B 0.000,C 90.000,E1 46.539} C_DIS
LIN {X 0.085,Y -568.682,Z 1007.054,A 0.000,B 0.000,C 90.000,E1 45.729} C_DIS
LIN {X 0.066,Y -566.744,Z 1007.048,A 0.000,B 0.000,C 90.000,E1 44.636} C_DIS
LIN {X 0.021,Y -564.494,Z 1007.042,A 0.000,B 0.000,C 90.000,E1 43.542} C_DIS
LIN {X -0.204,Y -563.280,Z 1007.039,A 0.000,B 0.000,C 90.000,E1 43.014} C_DIS
LIN {X 0.040,Y -561.150,Z 1007.034,A 0.000,B 0.000,C 90.000,E1 42.162} C_DIS
LIN {X 0.172,Y -559.631,Z 1007.031,A 0.000,B 0.000,C 90.000,E1 41.595} C_DIS
LIN {X 0.002,Y -556.984,Z 1007.027,A 0.000,B 0.000,C 90.000,E1 40.782} C_DIS
LIN {X 0.168,Y -554.095,Z 1007.022,A 0.000,B 0.000,C 90.000,E1 39.930} C_DIS
LIN {X 0.239,Y -553.121,Z 1007.020,A 0.000,B 0.000,C 90.000,E1 39.644} C_DIS
LIN {X -0.056,Y -550.917,Z 1007.017,A 0.000,B 0.000,C 90.000,E1 39.116} C_DIS
LIN {X -0.072,Y -545.442,Z 1007.010,A 0.000,B 0.000,C 90.000,E1 37.855} C_DIS
LIN {X -0.113,Y -540.692,Z 1007.005,A 0.000,B 0.000,C 90.000,E1 36.870} C_DIS
LIN {X -0.054,Y -536.422,Z 1007.000,A 0.000,B 0.000,C 90.000,E1 36.011} C_DIS
LIN {X -0.047,Y -531.851,Z 1006.995,A 0.000,B 0.000,C 90.000,E1 35.152} C_DIS
LIN {X 0.202,Y -527.814,Z 1006.991,A 0.000,B 0.000,C 90.000,E1 34.405} C_DIS
LIN {X -0.184,Y -522.641,Z 1006.987,A 0.000,B 0.000,C 90.000,E1 33.579} C_DIS
LIN {X -0.013,Y -518.043,Z 1006.982,A 0.000,B 0.000,C 90.000,E1 32.832} C_DIS
LIN {X 0.113,Y -513.070,Z 1006.978,A 0.000,B 0.000,C 90.000,E1 32.084} C_DIS
LIN {X 0.191,Y -507.771,Z 1006.974,A 0.000,B 0.000,C 90.000,E1 31.337} C_DIS
LIN {X -0.286,Y -503.107,Z 1006.971,A 0.000,B 0.000,C 90.000,E1 30.797} C_DIS
LIN {X -0.236,Y -498.219,Z 1006.968,A 0.000,B 0.000,C 90.000,E1 30.207} C_DIS
LIN {X -0.046,Y -491.822,Z 1006.964,A 0.000,B 0.000,C 90.000,E1 29.461} C_DIS
LIN {X 0.021,Y -484.972,Z 1006.960,A 0.000,B 0.000,C 90.000,E1 28.743} C_DIS
LIN {X 0.010,Y -476.406,Z 1006.955,A 0.000,B 0.000,C 90.000,E1 27.897} C_DIS
LIN {X -0.036,Y -467.673,Z 1006.950,A 0.000,B 0.000,C 90.000,E1 27.078} C_DIS
LIN {X 0.219,Y -457.182,Z 1006.945,A 0.000,B 0.000,C 90.000,E1 26.104} C_DIS
LIN {X 0.165,Y -445.063,Z 1006.940,A 0.000,B 0.000,C 90.000,E1 25.079} C_DIS
LIN {X 0.030,Y -428.451,Z 1006.931,A 0.000,B 0.000,C 90.000,E1 23.643} C_DIS
LIN {X 0.144,Y -418.067,Z 1006.926,A 0.000,B 0.000,C 90.000,E1 22.642} C_DIS
LIN {X -0.080,Y -403.618,Z 1006.917,A 0.000,B 0.000,C 90.000,E1 21.153} C_DIS
LIN {X 0.107,Y -398.112,Z 1006.914,A 0.000,B 0.000,C 90.000,E1 20.482} C_DIS
LIN {X 0.001,Y -395.019,Z 1006.912,A 0.000,B 0.000,C 90.000,E1 20.066} C_DIS
LIN {X -0.146,Y -392.584,Z 1006.909,A 0.000,B 0.000,C 90.000,E1 19.631} C_DIS
LIN {X -0.203,Y -390.908,Z 1006.906,A 0.000,B 0.000,C 90.000,E1 19.033} C_DIS
LIN {X 0.126,Y -390.514,Z 1006.902,A 0.000,B 0.000,C 90.000,E1 18.362} C_DIS
LIN {X -0.138,Y -391.037,Z 1006.897,A 0.000,B 0.000,C 90.000,E1 17.511} C_DIS
LIN {X 0.013,Y -394.661,Z 1006.878,A 0.000,B 0.000,C 90.000,E1 13.939} C_DIS
LIN {X -0.119,Y -401.718,Z 1006.850,A 0.000,B 0.000,C 90.000,E1 9.029} C_DIS
LIN {X 0.140,Y -408.277,Z 1006.831,A 0.000,B 0.000,C 90.000,E1 5.511} C_DIS
LIN {X 0.149,Y -412.014,Z 1006.821,A 0.000,B 0.000,C 90.000,E1 3.784} C_DIS
LIN {X 0.179,Y -415.904,Z 1006.812,A 0.000,B 0.000,C 90.000,E1 2.064} C_DIS
LIN {X -0.204,Y -417.375,Z 1006.809,A 0.000,B 0.000,C 90.000,E1 1.604} C_DIS
LIN {X -0.176,Y -419.524,Z 1006.806,A 0.000,B 0.000,C 90.000,E1 1.088} C_DIS
LIN {X -0.148,Y -421.700,Z 1006.804,A 0.000,B 0.000,C 90.000,E1 0.745} C_DIS
LIN {X 0.090,Y -423.459,Z 1006.803,A 0.000,B 0.000,C 90.000,E1 0.458} C_DIS
LIN {X -0.178,Y -426.944,Z 1006.801,A 0.000,B 0.000,C 90.000,E1 0.172} C_DIS
LIN {X 0.000,Y -428.893,Z 1006.800,A 0.000,B 0.000,C 90.000,E1 360.000} C_DIS
LIN {X -0.086,Y -435.820,Z 1006.798,A 0.000,B 0.000,C 90.000,E1 359.599} C_DIS
LIN {X -0.216,Y -442.302,Z 1006.796,A 0.000,B 0.000,C 90.000,E1 359.255} C_DIS
LIN {X -0.068,Y -458.836,Z 1006.790,A 0.000,B 0.000,C 90.000,E1 358.282} C_DIS
LIN {X 0.168,Y -472.037,Z 1006.786,A 0.000,B 0.000,C 90.000,E1 357.478} C_DIS
LIN {X -0.088,Y -483.589,Z 1006.782,A 0.000,B 0.000,C 90.000,E1 356.846} C_DIS
LIN {X -0.023,Y -495.125,Z 1006.779,A 0.000,B 0.000,C 90.000,E1 356.159} C_DIS
LIN {X -0.162,Y -504.809,Z 1006.775,A 0.000,B 0.000,C 90.000,E1 355.584} C_DIS
LIN {X -0.145,Y -511.210,Z 1006.773,A 0.000,B 0.000,C 90.000,E1 355.179} C_DIS
LIN {X 0.176,Y -517.333,Z 1006.771,A 0.000,B 0.000,C 90.000,E1 354.723} C_DIS
LIN {X -0.169,Y -524.830,Z 1006.768,A 0.000,B 0.000,C 90.000,E1 354.204} C_DIS
LIN {X -0.094,Y -531.941,Z 1006.765,A 0.000,B 0.000,C 90.000,E1 353.628} C_DIS
LIN {X 0.169,Y -537.618,Z 1006.762,A 0.000,B 0.000,C 90.000,E1 353.109} C_DIS
LIN {X 0.222,Y -544.368,Z 1006.758,A 0.000,B 0.000,C 90.000,E1 352.470} C_DIS
LIN {X -0.120,Y -550.729,Z 1006.755,A 0.000,B 0.000,C 90.000,E1 351.837} C_DIS
LIN {X 0.139,Y -555.623,Z 1006.752,A 0.000,B 0.000,C 90.000,E1 351.254} C_DIS
LIN {X 0.155,Y -561.160,Z 1006.748,A 0.000,B 0.000,C 90.000,E1 350.557} C_DIS
LIN {X 0.058,Y -564.334,Z 1006.745,A 0.000,B 0.000,C 90.000,E1 350.151} C_DIS
LIN {X 0.148,Y -568.808,Z 1006.742,A 0.000,B 0.000,C 90.000,E1 349.454} C_DIS
LIN {X -0.216,Y -575.302,Z 1006.735,A 0.000,B 0.000,C 90.000,E1 348.398} C_DIS
LIN {X -0.035,Y -579.003,Z 1006.732,A 0.000,B 0.000,C 90.000,E1 347.701} C_DIS
LIN {X -0.264,Y -584.463,Z 1006.726,A 0.000,B 0.000,C 90.000,E1 346.645} C_DIS
LIN {X 0.057,Y -590.173,Z 1006.719,A 0.000,B 0.000,C 90.000,E1 345.408} C_DIS
LIN {X -0.075,Y -593.216,Z 1006.715,A 0.000,B 0.000,C 90.000,E1 344.755} C_DIS
LIN {X -0.254,Y -596.699,Z 1006.711,A 0.000,B 0.000,C 90.000,E1 343.976} C_DIS
LIN {X 0.357,Y -602.131,Z 1006.704,A 0.000,B 0.000,C 90.000,E1 342.598} C_DIS
LIN {X -0.208,Y -604.303,Z 1006.701,A 0.000,B 0.000,C 90.000,E1 342.127} C_DIS
LIN {X 0.148,Y -609.270,Z 1006.693,A 0.000,B 0.000,C 90.000,E1 340.786} C_DIS
LIN {X 0.128,Y -612.154,Z 1006.689,A 0.000,B 0.000,C 90.000,E1 340.007} C_DIS
LIN {X 0.305,Y -615.462,Z 1006.683,A 0.000,B 0.000,C 90.000,E1 338.954} C_DIS
LIN {X -0.268,Y -618.583,Z 1006.678,A 0.000,B 0.000,C 90.000,E1 337.975} C_DIS
LIN {X -0.005,Y -622.335,Z 1006.670,A 0.000,B 0.000,C 90.000,E1 336.666} C_DIS
LIN {X -0.260,Y -624.394,Z 1006.666,A 0.000,B 0.000,C 90.000,E1 335.921} C_DIS
LIN {X 0.360,Y -627.534,Z 1006.659,A 0.000,B 0.000,C 90.000,E1 334.588} C_DIS
LIN {X 0.192,Y -630.450,Z 1006.652,A 0.000,B 0.000,C 90.000,E1 333.332} C_DIS
LIN {X -0.185,Y -633.383,Z 1006.644,A 0.000,B 0.000,C 90.000,E1 331.847} C_DIS
LIN {X -0.201,Y -635.985,Z 1006.635,A 0.000,B 0.000,C 90.000,E1 330.333} C_DIS
LIN {X -0.258,Y -637.578,Z 1006.630,A 0.000,B 0.000,C 90.000,E1 329.331} C_DIS
LIN {X -0.292,Y -638.965,Z 1006.624,A 0.000,B 0.000,C 90.000,E1 328.329} C_DIS
LIN {X 0.079,Y -640.497,Z 1006.617,A 0.000,B 0.000,C 90.000,E1 327.041} C_DIS
LIN {X 0.426,Y -641.581,Z 1006.611,A 0.000,B 0.000,C 90.000,E1 326.008} C_DIS
LIN {X -0.226,Y -642.603,Z 1006.604,A 0.000,B 0.000,C 90.000,E1 324.815} C_DIS
LIN {X 0.141,Y -643.149,Z 1006.599,A 0.000,B 0.000,C 90.000,E1 323.783} C_DIS
LIN {X -0.112,Y -643.714,Z 1006.592,A 0.000,B 0.000,C 90.000,E1 322.557} C_DIS
LIN {X -0.117,Y -644.343,Z 1006.581,A 0.000,B 0.000,C 90.000,E1 320.561} C_DIS
LIN {X 0.148,Y -645.578,Z 1006.566,A 0.000,B 0.000,C 90.000,E1 317.796} C_DIS
LIN {X 0.275,Y -646.259,Z 1006.559,A 0.000,B 0.000,C 90.000,E1 316.539} C_DIS
LIN {X -0.174,Y -647.200,Z 1006.549,A 0.000,B 0.000,C 90.000,E1 314.838} C_DIS
LIN {X -0.072,Y -648.178,Z 1006.541,A 0.000,B 0.000,C 90.000,E1 313.338} C_DIS
LIN {X 0.048,Y -649.106,Z 1006.533,A 0.000,B 0.000,C 90.000,E1 311.838} C_DIS
LIN {X -0.260,Y -649.931,Z 1006.524,A 0.000,B 0.000,C 90.000,E1 310.378} C_DIS
LIN {X -0.037,Y -650.596,Z 1006.515,A 0.000,B 0.000,C 90.000,E1 308.624} C_DIS
LIN {X 0.233,Y -651.074,Z 1006.508,A 0.000,B 0.000,C 90.000,E1 307.363} C_DIS
LIN {X 0.185,Y -651.342,Z 1006.502,A 0.000,B 0.000,C 90.000,E1 306.377} C_DIS
LIN {X 0.146,Y -651.508,Z 1006.497,A 0.000,B 0.000,C 90.000,E1 305.391} C_DIS
LIN {X 0.148,Y -652.019,Z 1006.484,A 0.000,B 0.000,C 90.000,E1 303.166} C_DIS
LIN {X -0.194,Y -655.199,Z 1006.461,A 0.000,B 0.000,C 90.000,E1 298.999} C_DIS
LIN {X 0.273,Y -657.993,Z 1006.449,A 0.000,B 0.000,C 90.000,E1 296.744} C_DIS
LIN {X 0.020,Y -659.672,Z 1006.442,A 0.000,B 0.000,C 90.000,E1 295.540} C_DIS
LIN {X -0.062,Y -660.887,Z 1006.437,A 0.000,B 0.000,C 90.000,E1 294.567} C_DIS
LIN {X -0.076,Y -661.759,Z 1006.431,A 0.000,B 0.000,C 90.000,E1 293.590} C_DIS
LIN {X 0.321,Y -662.214,Z 1006.427,A 0.000,B 0.000,C 90.000,E1 292.823} C_DIS
LIN {X -0.405,Y -662.439,Z 1006.423,A 0.000,B 0.000,C 90.000,E1 292.153} C_DIS
LIN {X -0.147,Y -662.045,Z 1006.420,A 0.000,B 0.000,C 90.000,E1 291.642} C_DIS
LIN {X -0.263,Y -661.717,Z 1006.419,A 0.000,B 0.000,C 90.000,E1 291.408} C_DIS
LIN {X -0.253,Y -660.597,Z 1006.416,A 0.000,B 0.000,C 90.000,E1 290.918} C_DIS
LIN {X -0.133,Y -659.469,Z 1006.415,A 0.000,B 0.000,C 90.000,E1 290.663} C_DIS
LIN {X -0.248,Y -657.745,Z 1006.413,A 0.000,B 0.000,C 90.000,E1 290.429} C_DIS
LIN {X -0.140,Y -656.268,Z 1006.412,A 0.000,B 0.000,C 90.000,E1 290.174} C_DIS
LIN {X -0.314,Y -655.119,Z 1006.411,A 0.000,B 0.000,C 90.000,E1 290.066} C_DIS
LIN {X 0.105,Y -650.327,Z 1006.410,A 0.000,B 0.000,C 90.000,E1 289.704} C_DIS
LIN {X -0.017,Y -648.525,Z 1006.409,A 0.000,B 0.000,C 90.000,E1 289.577} C_DIS
LIN {X -0.281,Y -641.764,Z 1006.407,A 0.000,B 0.000,C 90.000,E1 289.214} C_DIS
LIN {X 0.025,Y -635.367,Z 1006.405,A 0.000,B 0.000,C 90.000,E1 288.852} C_DIS
LIN {X -0.013,Y -634.178,Z 1006.404,A 0.000,B 0.000,C 90.000,E1 288.779} C_DIS
LIN {X 0.320,Y -632.410,Z 1006.404,A 0.000,B 0.000,C 90.000,E1 288.598} C_DIS
LIN {X 0.280,Y -632.376,Z 1006.404,A 0.000,B 0.000,C 90.000,E1 288.598} C_DIS
LIN {X -0.113,Y -632.313,Z 1006.403,A 0.000,B 0.000,C 90.000,E1 288.598} C_DIS
LIN {X -0.152,Y -632.327,Z 1006.403,A 0.000,B 0.000,C 90.000,E1 288.598} C_DIS
LIN {X -0.166,Y -634.115,Z 1006.401,A 0.000,B 0.000,C 90.000,E1 288.236} C_DIS
LIN {X -0.160,Y -638.716,Z 1006.397,A 0.000,B 0.000,C 90.000,E1 287.511} C_DIS
LIN {X -0.256,Y -640.402,Z 1006.396,A 0.000,B 0.000,C 90.000,E1 287.275} C_DIS
LIN {X 0.139,Y -644.891,Z 1006.392,A 0.000,B 0.000,C 90.000,E1 286.496} C_DIS
LIN {X -0.143,Y -648.162,Z 1006.388,A 0.000,B 0.000,C 90.000,E1 285.898} C_DIS
LIN {X 0.361,Y -649.835,Z 1006.386,A 0.000,B 0.000,C 90.000,E1 285.481} C_DIS
LIN {X 0.093,Y -651.721,Z 1006.383,A 0.000,B 0.000,C 90.000,E1 285.009} C_DIS
LIN {X -0.036,Y -652.612,Z 1006.382,A 0.000,B 0.000,C 90.000,E1 284.773} C_DIS
LIN {X 0.230,Y -654.487,Z 1006.378,A 0.000,B 0.000,C 90.000,E1 284.008} C_DIS
LIN {X -0.003,Y -655.401,Z 1006.375,A 0.000,B 0.000,C 90.000,E1 283.536} C_DIS
LIN {X 0.295,Y -656.185,Z 1006.371,A 0.000,B 0.000,C 90.000,E1 282.771} C_DIS
LIN {X 0.070,Y -656.491,Z 1006.368,A 0.000,B 0.000,C 90.000,E1 282.299} C_DIS
LIN {X -0.155,Y -656.533,Z 1006.366,A 0.000,B 0.000,C 90.000,E1 281.827} C_DIS
LIN {X 0.019,Y -656.183,Z 1006.362,A 0.000,B 0.000,C 90.000,E1 281.074} C_DIS
LIN {X -0.210,Y -655.637,Z 1006.359,A 0.000,B 0.000,C 90.000,E1 280.602} C_DIS
LIN {X 0.197,Y -654.795,Z 1006.356,A 0.000,B 0.000,C 90.000,E1 280.074} C_DIS
LIN {X -0.160,Y -653.697,Z 1006.353,A 0.000,B 0.000,C 90.000,E1 279.613} C_DIS
LIN {X -0.286,Y -653.053,Z 1006.352,A 0.000,B 0.000,C 90.000,E1 279.378} C_DIS
LIN {X -0.006,Y -651.477,Z 1006.349,A 0.000,B 0.000,C 90.000,E1 278.859} C_DIS
LIN {X 0.268,Y -649.502,Z 1006.346,A 0.000,B 0.000,C 90.000,E1 278.341} C_DIS
LIN {X -0.141,Y -646.528,Z 1006.343,A 0.000,B 0.000,C 90.000,E1 277.757} C_DIS
LIN {X -0.025,Y -642.486,Z 1006.340,A 0.000,B 0.000,C 90.000,E1 277.125} C_DIS
LIN {X 0.188,Y -638.623,Z 1006.337,A 0.000,B 0.000,C 90.000,E1 276.606} C_DIS
LIN {X -0.257,Y -634.191,Z 1006.334,A 0.000,B 0.000,C 90.000,E1 276.144} C_DIS
LIN {X -0.139,Y -627.994,Z 1006.331,A 0.000,B 0.000,C 90.000,E1 275.511} C_DIS
LIN {X 0.230,Y -622.648,Z 1006.328,A 0.000,B 0.000,C 90.000,E1 274.992} C_DIS
LIN {X 0.237,Y -618.489,Z 1006.326,A 0.000,B 0.000,C 90.000,E1 274.645} C_DIS
LIN {X -0.147,Y -612.553,Z 1006.324,A 0.000,B 0.000,C 90.000,E1 274.245} C_DIS
LIN {X -0.163,Y -606.242,Z 1006.321,A 0.000,B 0.000,C 90.000,E1 273.841} C_DIS
LIN {X -0.076,Y -598.501,Z 1006.319,A 0.000,B 0.000,C 90.000,E1 273.383} C_DIS
LIN {X 0.304,Y -591.718,Z 1006.317,A 0.000,B 0.000,C 90.000,E1 273.037} C_DIS
LIN {X -0.134,Y -584.481,Z 1006.316,A 0.000,B 0.000,C 90.000,E1 272.808} C_DIS
LIN {X -0.069,Y -578.674,Z 1006.315,A 0.000,B 0.000,C 90.000,E1 272.636} C_DIS
LIN {X -0.212,Y -570.940,Z 1006.314,A 0.000,B 0.000,C 90.000,E1 272.465} C_DIS
LIN {X 0.079,Y -566.066,Z 1006.313,A 0.000,B 0.000,C 90.000,E1 272.350} C_DIS
LIN {X 0.177,Y -561.326,Z 1006.313,A 0.000,B 0.000,C 90.000,E1 272.293} C_DIS
LIN {X -0.021,Y -558.482,Z 1006.313,A 0.000,B 0.000,C 90.000,E1 272.293} C_DIS
LIN {X -0.061,Y -543.659,Z 1006.313,A 0.000,B 0.000,C 90.000,E1 272.293} C_DIS
LIN {X -0.227,Y -542.955,Z 1006.312,A 0.000,B 0.000,C 90.000,E1 272.178} C_DIS
LIN {X -0.201,Y -542.147,Z 1006.308,A 0.000,B 0.000,C 90.000,E1 271.432} C_DIS
LIN {X -0.022,Y -540.834,Z 1006.297,A 0.000,B 0.000,C 90.000,E1 269.427} C_DIS
LIN {X 0.117,Y -539.712,Z 1006.287,A 0.000,B 0.000,C 90.000,E1 267.707} C_DIS
LIN {X 0.269,Y -538.196,Z 1006.276,A 0.000,B 0.000,C 90.000,E1 265.698} C_DIS
LIN {X -0.166,Y -536.823,Z 1006.267,A 0.000,B 0.000,C 90.000,E1 264.033} C_DIS
LIN {X -0.039,Y -535.571,Z 1006.259,A 0.000,B 0.000,C 90.000,E1 262.591} C_DIS
LIN {X 0.140,Y -534.196,Z 1006.251,A 0.000,B 0.000,C 90.000,E1 261.141} C_DIS
LIN {X -0.277,Y -532.993,Z 1006.245,A 0.000,B 0.000,C 90.000,E1 260.038} C_DIS
LIN {X 0.035,Y -530.779,Z 1006.233,A 0.000,B 0.000,C 90.000,E1 257.993} C_DIS
LIN {X -0.299,Y -529.262,Z 1006.225,A 0.000,B 0.000,C 90.000,E1 256.589} C_DIS
LIN {X -0.082,Y -528.330,Z 1006.221,A 0.000,B 0.000,C 90.000,E1 255.700} C_DIS
LIN {X -0.171,Y -525.995,Z 1006.209,A 0.000,B 0.000,C 90.000,E1 253.685} C_DIS
LIN {X -0.177,Y -524.458,Z 1006.201,A 0.000,B 0.000,C 90.000,E1 252.236} C_DIS
LIN {X 0.131,Y -523.117,Z 1006.195,A 0.000,B 0.000,C 90.000,E1 251.040} C_DIS
LIN {X -0.090,Y -520.860,Z 1006.185,A 0.000,B 0.000,C 90.000,E1 249.316} C_DIS
LIN {X 0.134,Y -518.624,Z 1006.175,A 0.000,B 0.000,C 90.000,E1 247.539} C_DIS
LIN {X 0.221,Y -517.022,Z 1006.169,A 0.000,B 0.000,C 90.000,E1 246.357} C_DIS
LIN {X 0.280,Y -514.446,Z 1006.159,A 0.000,B 0.000,C 90.000,E1 244.588} C_DIS
LIN {X 0.055,Y -512.567,Z 1006.153,A 0.000,B 0.000,C 90.000,E1 243.435} C_DIS
LIN {X -0.196,Y -510.678,Z 1006.146,A 0.000,B 0.000,C 90.000,E1 242.281} C_DIS
LIN {X -0.152,Y -508.300,Z 1006.138,A 0.000,B 0.000,C 90.000,E1 240.795} C_DIS
LIN {X 0.022,Y -506.235,Z 1006.131,A 0.000,B 0.000,C 90.000,E1 239.587} C_DIS
LIN {X -0.092,Y -504.030,Z 1006.124,A 0.000,B 0.000,C 90.000,E1 238.408} C_DIS
LIN {X -0.108,Y -501.042,Z 1006.116,A 0.000,B 0.000,C 90.000,E1 236.914} C_DIS
LIN {X -0.061,Y -499.077,Z 1006.111,A 0.000,B 0.000,C 90.000,E1 236.008} C_DIS
LIN {X -0.164,Y -496.465,Z 1006.104,A 0.000,B 0.000,C 90.000,E1 234.815} C_DIS
LIN {X 0.097,Y -492.025,Z 1006.094,A 0.000,B 0.000,C 90.000,E1 232.970} C_DIS
LIN {X 0.002,Y -486.848,Z 1006.083,A 0.000,B 0.000,C 90.000,E1 230.848} C_DIS
LIN {X -0.002,Y -484.000,Z 1006.076,A 0.000,B 0.000,C 90.000,E1 229.622} C_DIS
LIN {X 0.014,Y -480.426,Z 1006.067,A 0.000,B 0.000,C 90.000,E1 228.081} C_DIS
LIN {X -0.036,Y -475.167,Z 1006.053,A 0.000,B 0.000,C 90.000,E1 225.607} C_DIS
LIN {X 0.224,Y -471.342,Z 1006.043,A 0.000,B 0.000,C 90.000,E1 223.704} C_DIS
LIN {X 0.003,Y -468.010,Z 1006.034,A 0.000,B 0.000,C 90.000,E1 222.162} C_DIS
LIN {X 0.136,Y -463.855,Z 1006.024,A 0.000,B 0.000,C 90.000,E1 220.253} C_DIS
LIN {X -0.136,Y -459.525,Z 1006.013,A 0.000,B 0.000,C 90.000,E1 218.382} C_DIS
LIN {X -0.163,Y -456.061,Z 1006.004,A 0.000,B 0.000,C 90.000,E1 216.790} C_DIS
LIN {X 0.189,Y -451.842,Z 1005.994,A 0.000,B 0.000,C 90.000,E1 214.818} C_DIS
LIN {X 0.254,Y -446.931,Z 1005.981,A 0.000,B 0.000,C 90.000,E1 212.546} C_DIS
LIN {X 0.094,Y -441.957,Z 1005.968,A 0.000,B 0.000,C 90.000,E1 210.285} C_DIS
LIN {X -0.139,Y -439.813,Z 1005.963,A 0.000,B 0.000,C 90.000,E1 209.333} C_DIS
LIN {X 0.057,Y -434.551,Z 1005.950,A 0.000,B 0.000,C 90.000,E1 207.001} C_DIS
LIN {X -0.086,Y -430.052,Z 1005.939,A 0.000,B 0.000,C 90.000,E1 205.027} C_DIS
LIN {X 0.080,Y -426.271,Z 1005.930,A 0.000,B 0.000,C 90.000,E1 203.334} C_DIS
LIN {X 0.078,Y -419.697,Z 1005.913,A 0.000,B 0.000,C 90.000,E1 200.301} C_DIS
LIN {X -0.103,Y -415.038,Z 1005.900,A 0.000,B 0.000,C 90.000,E1 197.946} C_DIS
LIN {X -0.132,Y -410.791,Z 1005.886,A 0.000,B 0.000,C 90.000,E1 195.552} C_DIS
LIN {X 0.012,Y -406.383,Z 1005.871,A 0.000,B 0.000,C 90.000,E1 192.771} C_DIS
LIN {X 0.220,Y -403.276,Z 1005.859,A 0.000,B 0.000,C 90.000,E1 190.658} C_DIS
LIN {X -0.179,Y -401.843,Z 1005.854,A 0.000,B 0.000,C 90.000,E1 189.670} C_DIS
LIN {X 0.198,Y -400.830,Z 1005.848,A 0.000,B 0.000,C 90.000,E1 188.568} C_DIS
LIN {X 0.112,Y -400.709,Z 1005.842,A 0.000,B 0.000,C 90.000,E1 187.530} C_DIS
LIN {X 0.101,Y -400.872,Z 1005.840,A 0.000,B 0.000,C 90.000,E1 187.182} C_DIS
LIN {X 0.075,Y -402.218,Z 1005.836,A 0.000,B 0.000,C 90.000,E1 186.486} C_DIS
LIN {X 0.019,Y -402.687,Z 1005.834,A 0.000,B 0.000,C 90.000,E1 186.144} C_DIS
LIN {X 0.036,Y -403.047,Z 1005.833,A 0.000,B 0.000,C 90.000,E1 185.967} C_DIS
LIN {X 0.042,Y -404.523,Z 1005.831,A 0.000,B 0.000,C 90.000,E1 185.568} C_DIS
LIN {X 0.037,Y -405.952,Z 1005.829,A 0.000,B 0.000,C 90.000,E1 185.220} C_DIS
LIN {X 0.003,Y -407.708,Z 1005.827,A 0.000,B 0.000,C 90.000,E1 184.878} C_DIS
LIN {X -0.155,Y -410.711,Z 1005.824,A 0.000,B 0.000,C 90.000,E1 184.416} C_DIS
LIN {X -0.090,Y -414.596,Z 1005.822,A 0.000,B 0.000,C 90.000,E1 183.898} C_DIS
LIN {X -0.113,Y -424.304,Z 1005.815,A 0.000,B 0.000,C 90.000,E1 182.751} C_DIS
LIN {X 0.102,Y -431.343,Z 1005.811,A 0.000,B 0.000,C 90.000,E1 181.949} C_DIS
LIN {X 0.096,Y -442.515,Z 1005.804,A 0.000,B 0.000,C 90.000,E1 180.688} C_DIS
LIN {X -0.073,Y -454.813,Z 1005.796,A 0.000,B 0.000,C 90.000,E1 179.312} C_DIS
LIN {X -0.174,Y -462.831,Z 1005.791,A 0.000,B 0.000,C 90.000,E1 178.396} C_DIS
LIN {X 0.039,Y -469.385,Z 1005.787,A 0.000,B 0.000,C 90.000,E1 177.593} C_DIS
LIN {X 0.193,Y -478.097,Z 1005.781,A 0.000,B 0.000,C 90.000,E1 176.502} C_DIS
LIN {X -0.183,Y -482.978,Z 1005.777,A 0.000,B 0.000,C 90.000,E1 175.927} C_DIS
LIN {X -0.064,Y -490.835,Z 1005.771,A 0.000,B 0.000,C 90.000,E1 174.837} C_DIS
LIN {X -0.185,Y -496.188,Z 1005.767,A 0.000,B 0.000,C 90.000,E1 174.090} C_DIS
LIN {X 0.151,Y -503.401,Z 1005.761,A 0.000,B 0.000,C 90.000,E1 172.996} C_DIS
LIN {X 0.205,Y -508.302,Z 1005.757,A 0.000,B 0.000,C 90.000,E1 172.243} C_DIS
LIN {X -0.158,Y -511.332,Z 1005.755,A 0.000,B 0.000,C 90.000,E1 171.837} C_DIS
LIN {X 0.016,Y -519.610,Z 1005.747,A 0.000,B 0.000,C 90.000,E1 170.500} C_DIS
LIN {X 0.277,Y -529.231,Z 1005.738,A 0.000,B 0.000,C 90.000,E1 168.870} C_DIS
LIN {X 0.205,Y -538.599,Z 1005.730,A 0.000,B 0.000,C 90.000,E1 167.297} C_DIS
LIN {X 0.091,Y -545.140,Z 1005.723,A 0.000,B 0.000,C 90.000,E1 166.172} C_DIS
LIN {X -0.027,Y -550.029,Z 1005.719,A 0.000,B 0.000,C 90.000,E1 165.338} C_DIS
LIN {X 0.031,Y -556.284,Z 1005.712,A 0.000,B 0.000,C 90.000,E1 164.212} C_DIS
LIN {X 0.171,Y -562.330,Z 1005.706,A 0.000,B 0.000,C 90.000,E1 163.087} C_DIS
LIN {X 0.072,Y -570.140,Z 1005.698,A 0.000,B 0.000,C 90.000,E1 161.583} C_DIS
LIN {X -0.145,Y -574.285,Z 1005.693,A 0.000,B 0.000,C 90.000,E1 160.786} C_DIS
LIN {X -0.212,Y -580.165,Z 1005.686,A 0.000,B 0.000,C 90.000,E1 159.571} C_DIS
LIN {X 0.016,Y -585.716,Z 1005.680,A 0.000,B 0.000,C 90.000,E1 158.337} C_DIS
LIN {X -0.158,Y -590.310,Z 1005.674,A 0.000,B 0.000,C 90.000,E1 157.283} C_DIS
LIN {X -0.174,Y -593.557,Z 1005.669,A 0.000,B 0.000,C 90.000,E1 156.485} C_DIS
LIN {X 0.172,Y -595.604,Z 1005.666,A 0.000,B 0.000,C 90.000,E1 155.921} C_DIS
LIN {X 0.368,Y -599.345,Z 1005.661,A 0.000,B 0.000,C 90.000,E1 154.845} C_DIS
LIN {X 0.146,Y -601.996,Z 1005.656,A 0.000,B 0.000,C 90.000,E1 154.076} C_DIS
LIN {X -0.165,Y -605.952,Z 1005.649,A 0.000,B 0.000,C 90.000,E1 152.794} C_DIS
LIN {X 0.363,Y -610.494,Z 1005.640,A 0.000,B 0.000,C 90.000,E1 151.179} C_DIS
LIN {X -0.059,Y -614.040,Z 1005.633,A 0.000,B 0.000,C 90.000,E1 149.921} C_DIS
LIN {X 0.132,Y -616.926,Z 1005.627,A 0.000,B 0.000,C 90.000,E1 148.869} C_DIS
LIN {X 0.110,Y -621.032,Z 1005.619,A 0.000,B 0.000,C 90.000,E1 147.327} C_DIS
LIN {X -0.031,Y -625.826,Z 1005.609,A 0.000,B 0.000,C 90.000,E1 145.548} C_DIS
LIN {X -0.223,Y -630.633,Z 1005.599,A 0.000,B 0.000,C 90.000,E1 143.783} C_DIS
LIN {X -0.300,Y -634.600,Z 1005.590,A 0.000,B 0.000,C 90.000,E1 142.271} C_DIS
LIN {X -0.176,Y -637.278,Z 1005.585,A 0.000,B 0.000,C 90.000,E1 141.251} C_DIS
LIN {X -0.119,Y -640.530,Z 1005.578,A 0.000,B 0.000,C 90.000,E1 139.989} C_DIS
LIN {X -0.013,Y -643.727,Z 1005.571,A 0.000,B 0.000,C 90.000,E1 138.728} C_DIS
LIN {X -0.043,Y -648.227,Z 1005.561,A 0.000,B 0.000,C 90.000,E1 136.986} C_DIS
LIN {X 0.095,Y -652.364,Z 1005.553,A 0.000,B 0.000,C 90.000,E1 135.486} C_DIS
LIN {X 0.177,Y -660.708,Z 1005.538,A 0.000,B 0.000,C 90.000,E1 132.771} C_DIS
LIN {X 0.108,Y -666.334,Z 1005.528,A 0.000,B 0.000,C 90.000,E1 131.067} C_DIS
LIN {X 0.150,Y -670.283,Z 1005.521,A 0.000,B 0.000,C 90.000,E1 129.850} C_DIS
LIN {X -0.183,Y -673.239,Z 1005.516,A 0.000,B 0.000,C 90.000,E1 128.910} C_DIS
LIN {X -0.056,Y -676.031,Z 1005.511,A 0.000,B 0.000,C 90.000,E1 127.935} C_DIS
LIN {X -0.161,Y -680.160,Z 1005.503,A 0.000,B 0.000,C 90.000,E1 126.503} C_DIS
LIN {X 0.367,Y -684.066,Z 1005.495,A 0.000,B 0.000,C 90.000,E1 125.025} C_DIS
LIN {X 0.005,Y -687.272,Z 1005.488,A 0.000,B 0.000,C 90.000,E1 123.865} C_DIS
LIN {X -0.148,Y -689.119,Z 1005.484,A 0.000,B 0.000,C 90.000,E1 123.166} C_DIS
LIN {X 0.392,Y -693.280,Z 1005.475,A 0.000,B 0.000,C 90.000,E1 121.465} C_DIS
LIN {X 0.163,Y -695.650,Z 1005.470,A 0.000,B 0.000,C 90.000,E1 120.541} C_DIS
LIN {X -0.034,Y -697.638,Z 1005.465,A 0.000,B 0.000,C 90.000,E1 119.617} C_DIS
LIN {X -0.207,Y -699.204,Z 1005.459,A 0.000,B 0.000,C 90.000,E1 118.693} C_DIS
LIN {X 0.251,Y -700.446,Z 1005.454,A 0.000,B 0.000,C 90.000,E1 117.719} C_DIS
LIN {X 0.257,Y -701.926,Z 1005.444,A 0.000,B 0.000,C 90.000,E1 115.848} C_DIS
LIN {X -0.203,Y -702.602,Z 1005.439,A 0.000,B 0.000,C 90.000,E1 114.951} C_DIS
LIN {X 0.339,Y -702.785,Z 1005.435,A 0.000,B 0.000,C 90.000,E1 114.207} C_DIS
LIN {X -0.024,Y -702.593,Z 1005.433,A 0.000,B 0.000,C 90.000,E1 114.003} C_DIS
LIN {X 0.245,Y -701.849,Z 1005.431,A 0.000,B 0.000,C 90.000,E1 113.515} C_DIS
LIN {X -0.130,Y -699.879,Z 1005.428,A 0.000,B 0.000,C 90.000,E1 113.078} C_DIS
LIN {X 0.137,Y -698.725,Z 1005.427,A 0.000,B 0.000,C 90.000,E1 112.823} C_DIS
LIN {X -0.002,Y -697.753,Z 1005.426,A 0.000,B 0.000,C 90.000,E1 112.717} C_DIS
LIN {X -0.264,Y -694.878,Z 1005.425,A 0.000,B 0.000,C 90.000,E1 112.514} C_DIS
LIN {X -0.159,Y -690.355,Z 1005.423,A 0.000,B 0.000,C 90.000,E1 112.206} C_DIS
LIN {X 0.253,Y -688.058,Z 1005.423,A 0.000,B 0.000,C 90.000,E1 112.078} C_DIS
LIN {X -0.231,Y -685.279,Z 1005.422,A 0.000,B 0.000,C 90.000,E1 112.025} C_DIS
LIN {X -0.010,Y -682.846,Z 1005.422,A 0.000,B 0.000,C 90.000,E1 111.950} C_DIS
LIN {X -0.021,Y -674.785,Z 1005.421,A 0.000,B 0.000,C 90.000,E1 111.844} C_DIS
LIN {X -0.080,Y -618.261,Z 1005.421,A 0.000,B 0.000,C 90.000,E1 111.844} C_DIS
LIN {X -0.194,Y -614.561,Z 1005.421,A 0.000,B 0.000,C 90.000,E1 111.770} C_DIS
LIN {X -0.031,Y -611.092,Z 1005.420,A 0.000,B 0.000,C 90.000,E1 111.663} C_DIS
LIN {X 0.160,Y -606.093,Z 1005.419,A 0.000,B 0.000,C 90.000,E1 111.461} C_DIS
LIN {X 0.047,Y -600.434,Z 1005.418,A 0.000,B 0.000,C 90.000,E1 111.227} C_DIS
LIN {X 0.231,Y -595.363,Z 1005.416,A 0.000,B 0.000,C 90.000,E1 110.918} C_DIS
LIN {X 0.204,Y -589.057,Z 1005.414,A 0.000,B 0.000,C 90.000,E1 110.482} C_DIS
LIN {X -0.107,Y -576.613,Z 1005.408,A 0.000,B 0.000,C 90.000,E1 109.504} C_DIS
LIN {X 0.145,Y -572.302,Z 1005.406,A 0.000,B 0.000,C 90.000,E1 109.141} C_DIS
LIN {X -0.053,Y -563.950,Z 1005.404,A 0.000,B 0.000,C 90.000,E1 108.671} C_DIS
LIN {X 0.205,Y -550.204,Z 1005.400,A 0.000,B 0.000,C 90.000,E1 107.946} C_DIS
LIN {X -0.186,Y -548.746,Z 1005.399,A 0.000,B 0.000,C 90.000,E1 107.819} C_DIS
LIN {X -0.228,Y -548.737,Z 1005.399,A 0.000,B 0.000,C 90.000,E1 107.819} C_DIS
LIN {X 0.198,Y -548.380,Z 1005.397,A 0.000,B 0.000,C 90.000,E1 107.511} C_DIS
LIN {X 0.105,Y -548.541,Z 1005.393,A 0.000,B 0.000,C 90.000,E1 106.677} C_DIS
LIN {X -0.170,Y -549.162,Z 1005.385,A 0.000,B 0.000,C 90.000,E1 105.300} C_DIS
LIN {X 0.164,Y -550.201,Z 1005.374,A 0.000,B 0.000,C 90.000,E1 103.300} C_DIS
LIN {X -0.070,Y -553.116,Z 1005.355,A 0.000,B 0.000,C 90.000,E1 99.962} C_DIS
LIN {X 0.025,Y -555.012,Z 1005.346,A 0.000,B 0.000,C 90.000,E1 98.276} C_DIS
LIN {X -0.052,Y -556.496,Z 1005.338,A 0.000,B 0.000,C 90.000,E1 96.891} C_DIS
LIN {X -0.160,Y -557.827,Z 1005.331,A 0.000,B 0.000,C 90.000,E1 95.511} C_DIS
LIN {X -0.238,Y -558.853,Z 1005.323,A 0.000,B 0.000,C 90.000,E1 94.131} C_DIS
LIN {X 0.253,Y -559.693,Z 1005.315,A 0.000,B 0.000,C 90.000,E1 92.694} C_DIS
LIN {X -0.209,Y -560.577,Z 1005.304,A 0.000,B 0.000,C 90.000,E1 90.802} C_DIS
LIN {X 0.269,Y -561.253,Z 1005.297,A 0.000,B 0.000,C 90.000,E1 89.370} C_DIS
LIN {X 0.094,Y -561.730,Z 1005.291,A 0.000,B 0.000,C 90.000,E1 88.282} C_DIS
LIN {X 0.038,Y -561.990,Z 1005.283,A 0.000,B 0.000,C 90.000,E1 86.906} C_DIS
LIN {X 0.020,Y -562.130,Z 1005.275,A 0.000,B 0.000,C 90.000,E1 85.527} C_DIS
LIN {X 0.009,Y -562.404,Z 1005.268,A 0.000,B 0.000,C 90.000,E1 84.147} C_DIS
LIN {X -0.266,Y -562.740,Z 1005.257,A 0.000,B 0.000,C 90.000,E1 82.243} C_DIS
LIN {X -0.126,Y -563.115,Z 1005.249,A 0.000,B 0.000,C 90.000,E1 80.849} C_DIS
LIN {X -0.203,Y -563.835,Z 1005.238,A 0.000,B 0.000,C 90.000,E1 78.926} C_DIS
LIN {X -0.152,Y -564.807,Z 1005.228,A 0.000,B 0.000,C 90.000,E1 76.992} C_DIS
LIN {X 0.049,Y -566.000,Z 1005.217,A 0.000,B 0.000,C 90.000,E1 75.046} C_DIS
LIN {X -0.127,Y -567.395,Z 1005.206,A 0.000,B 0.000,C 90.000,E1 73.142} C_DIS
LIN {X -0.066,Y -568.451,Z 1005.199,A 0.000,B 0.000,C 90.000,E1 71.764} C_DIS
LIN {X -0.001,Y -569.644,Z 1005.190,A 0.000,B 0.000,C 90.000,E1 70.115} C_DIS
LIN {X -0.082,Y -570.786,Z 1005.179,A 0.000,B 0.000,C 90.000,E1 68.209} C_DIS
LIN {X -0.107,Y -571.477,Z 1005.171,A 0.000,B 0.000,C 90.000,E1 66.847} C_DIS
LIN {X 0.035,Y -572.008,Z 1005.165,A 0.000,B 0.000,C 90.000,E1 65.741} C_DIS
LIN {X -0.272,Y -572.575,Z 1005.158,A 0.000,B 0.000,C 90.000,E1 64.409} C_DIS
LIN {X 0.037,Y -573.129,Z 1005.149,A 0.000,B 0.000,C 90.000,E1 62.743} C_DIS
LIN {X -0.155,Y -573.611,Z 1005.140,A 0.000,B 0.000,C 90.000,E1 61.129} C_DIS
LIN {X 0.095,Y -574.020,Z 1005.132,A 0.000,B 0.000,C 90.000,E1 59.744} C_DIS
LIN {X -0.141,Y -574.297,Z 1005.124,A 0.000,B 0.000,C 90.000,E1 58.408} C_DIS
LIN {X -0.208,Y -574.441,Z 1005.118,A 0.000,B 0.000,C 90.000,E1 57.327} C_DIS
LIN {X -0.135,Y -574.691,Z 1005.111,A 0.000,B 0.000,C 90.000,E1 55.960} C_DIS
LIN {X 0.116,Y -574.767,Z 1005.105,A 0.000,B 0.000,C 90.000,E1 54.848} C_DIS
LIN {X 0.049,Y -574.653,Z 1005.097,A 0.000,B 0.000,C 90.000,E1 53.497} C_DIS
LIN {X 0.033,Y -574.477,Z 1005.093,A 0.000,B 0.000,C 90.000,E1 52.683} C_DIS
LIN {X -0.186,Y -574.004,Z 1005.087,A 0.000,B 0.000,C 90.000,E1 51.618} C_DIS
LIN {X -0.061,Y -573.395,Z 1005.081,A 0.000,B 0.000,C 90.000,E1 50.517} C_DIS
LIN {X -0.386,Y -572.648,Z 1005.075,A 0.000,B 0.000,C 90.000,E1 49.461} C_DIS
LIN {X 0.086,Y -571.713,Z 1005.069,A 0.000,B 0.000,C 90.000,E1 48.324} C_DIS
LIN {X -0.003,Y -570.867,Z 1005.064,A 0.000,B 0.000,C 90.000,E1 47.514} C_DIS
LIN {X -0.065,Y -569.838,Z 1005.059,A 0.000,B 0.000,C 90.000,E1 46.701} C_DIS
LIN {X -0.167,Y -568.606,Z 1005.055,A 0.000,B 0.000,C 90.000,E1 45.891} C_DIS
LIN {X -0.279,Y -567.163,Z 1005.050,A 0.000,B 0.000,C 90.000,E1 45.081} C_DIS
LIN {X -0.009,Y -565.561,Z 1005.046,A 0.000,B 0.000,C 90.000,E1 44.231} C_DIS
LIN {X -0.071,Y -563.230,Z 1005.040,A 0.000,B 0.000,C 90.000,E1 43.137} C_DIS
LIN {X 0.165,Y -561.113,Z 1005.035,A 0.000,B 0.000,C 90.000,E1 42.285} C_DIS
LIN {X -0.078,Y -559.591,Z 1005.032,A 0.000,B 0.000,C 90.000,E1 41.757} C_DIS
LIN {X 0.197,Y -556.024,Z 1005.026,A 0.000,B 0.000,C 90.000,E1 40.620} C_DIS
LIN {X -0.077,Y -554.087,Z 1005.023,A 0.000,B 0.000,C 90.000,E1 40.092} C_DIS
LIN {X 0.063,Y -551.993,Z 1005.020,A 0.000,B 0.000,C 90.000,E1 39.519} C_DIS
LIN {X -0.034,Y -549.093,Z 1005.016,A 0.000,B 0.000,C 90.000,E1 38.830} C_DIS
LIN {X -0.268,Y -544.097,Z 1005.010,A 0.000,B 0.000,C 90.000,E1 37.729} C_DIS
LIN {X 0.003,Y -539.274,Z 1005.004,A 0.000,B 0.000,C 90.000,E1 36.710} C_DIS
LIN {X 0.041,Y -534.876,Z 1004.999,A 0.000,B 0.000,C 90.000,E1 35.851} C_DIS
LIN {X 0.301,Y -529.424,Z 1004.994,A 0.000,B 0.000,C 90.000,E1 34.818} C_DIS
LIN {X 0.094,Y -525.226,Z 1004.990,A 0.000,B 0.000,C 90.000,E1 34.119} C_DIS
LIN {X -0.271,Y -521.686,Z 1004.986,A 0.000,B 0.000,C 90.000,E1 33.579} C_DIS
LIN {X 0.061,Y -517.977,Z 1004.983,A 0.000,B 0.000,C 90.000,E1 32.959} C_DIS
LIN {X 0.184,Y -513.012,Z 1004.979,A 0.000,B 0.000,C 90.000,E1 32.212} C_DIS
LIN {X 0.260,Y -507.735,Z 1004.975,A 0.000,B 0.000,C 90.000,E1 31.465} C_DIS
LIN {X -0.219,Y -503.162,Z 1004.972,A 0.000,B 0.000,C 90.000,E1 30.924} C_DIS
LIN {X -0.293,Y -498.185,Z 1004.968,A 0.000,B 0.000,C 90.000,E1 30.335} C_DIS
LIN {X 0.157,Y -491.506,Z 1004.964,A 0.000,B 0.000,C 90.000,E1 29.539} C_DIS
LIN {X -0.098,Y -486.071,Z 1004.961,A 0.000,B 0.000,C 90.000,E1 28.999} C_DIS
LIN {X -0.036,Y -481.857,Z 1004.959,A 0.000,B 0.000,C 90.000,E1 28.565} C_DIS
LIN {X -0.082,Y -474.917,Z 1004.955,A 0.000,B 0.000,C 90.000,E1 27.897} C_DIS
LIN {X -0.089,Y -466.218,Z 1004.950,A 0.000,B 0.000,C 90.000,E1 27.078} C_DIS
LIN {X 0.196,Y -455.683,Z 1004.945,A 0.000,B 0.000,C 90.000,E1 26.104} C_DIS
LIN {X 0.212,Y -445.171,Z 1004.940,A 0.000,B 0.000,C 90.000,E1 25.207} C_DIS
LIN {X 0.068,Y -428.534,Z 1004.932,A 0.000,B 0.000,C 90.000,E1 23.770} C_DIS
LIN {X 0.018,Y -415.363,Z 1004.925,A 0.000,B 0.000,C 90.000,E1 22.514} C_DIS
LIN {X 0.164,Y -401.154,Z 1004.917,A 0.000,B 0.000,C 90.000,E1 20.972} C_DIS
LIN {X 0.159,Y -398.507,Z 1004.915,A 0.000,B 0.000,C 90.000,E1 20.663} C_DIS
LIN {X 0.026,Y -395.406,Z 1004.913,A 0.000,B 0.000,C 90.000,E1 20.248} C_DIS
LIN {X 0.061,Y -394.305,Z 1004.912,A 0.000,B 0.000,C 90.000,E1 20.066} C_DIS
LIN {X 0.127,Y -392.527,Z 1004.910,A 0.000,B 0.000,C 90.000,E1 19.704} C_DIS
LIN {X -0.192,Y -391.417,Z 1004.908,A 0.000,B 0.000,C 90.000,E1 19.396} C_DIS
LIN {X -0.167,Y -390.938,Z 1004.907,A 0.000,B 0.000,C 90.000,E1 19.214} C_DIS
LIN {X -0.030,Y -390.457,Z 1004.903,A 0.000,B 0.000,C 90.000,E1 18.489} C_DIS
LIN {X -0.142,Y -391.011,Z 1004.898,A 0.000,B 0.000,C 90.000,E1 17.583} C_DIS
LIN {X 0.026,Y -394.633,Z 1004.878,A 0.000,B 0.000,C 90.000,E1 14.008} C_DIS
LIN {X -0.070,Y -401.104,Z 1004.852,A 0.000,B 0.000,C 90.000,E1 9.443} C_DIS
LIN {X -0.135,Y -407.518,Z 1004.833,A 0.000,B 0.000,C 90.000,E1 5.967} C_DIS
LIN {X -0.164,Y -411.957,Z 1004.822,A 0.000,B 0.000,C 90.000,E1 3.898} C_DIS
LIN {X -0.127,Y -416.645,Z 1004.810,A 0.000,B 0.000,C 90.000,E1 1.835} C_DIS
LIN {X -0.099,Y -417.690,Z 1004.808,A 0.000,B 0.000,C 90.000,E1 1.489} C_DIS
LIN {X -0.068,Y -419.804,Z 1004.805,A 0.000,B 0.000,C 90.000,E1 0.974} C_DIS
LIN {X 0.209,Y -423.849,Z 1004.802,A 0.000,B 0.000,C 90.000,E1 0.344} C_DIS
LIN {X 0.000,Y -427.963,Z 1004.800,A 0.000,B 0.000,C 90.000,E1 360.000} C_DIS
LIN {X -0.179,Y -432.767,Z 1004.798,A 0.000,B 0.000,C 90.000,E1 359.714} C_DIS
LIN {X -0.113,Y -440.911,Z 1004.796,A 0.000,B 0.000,C 90.000,E1 359.255} C_DIS
LIN {X 0.005,Y -457.586,Z 1004.791,A 0.000,B 0.000,C 90.000,E1 358.282} C_DIS
LIN {X 0.003,Y -467.469,Z 1004.787,A 0.000,B 0.000,C 90.000,E1 357.707} C_DIS
LIN {X -0.043,Y -482.473,Z 1004.782,A 0.000,B 0.000,C 90.000,E1 356.846} C_DIS
LIN {X 0.101,Y -493.968,Z 1004.779,A 0.000,B 0.000,C 90.000,E1 356.159} C_DIS
LIN {X -0.259,Y -506.854,Z 1004.774,A 0.000,B 0.000,C 90.000,E1 355.412} C_DIS
LIN {X 0.038,Y -510.110,Z 1004.773,A 0.000,B 0.000,C 90.000,E1 355.179} C_DIS
LIN {X -0.034,Y -516.099,Z 1004.771,A 0.000,B 0.000,C 90.000,E1 354.780} C_DIS
LIN {X 0.170,Y -523.693,Z 1004.768,A 0.000,B 0.000,C 90.000,E1 354.204} C_DIS
LIN {X 0.163,Y -531.041,Z 1004.765,A 0.000,B 0.000,C 90.000,E1 353.628} C_DIS
LIN {X -0.140,Y -538.082,Z 1004.761,A 0.000,B 0.000,C 90.000,E1 353.053} C_DIS
LIN {X -0.010,Y -543.548,Z 1004.759,A 0.000,B 0.000,C 90.000,E1 352.534} C_DIS
LIN {X -0.273,Y -549.993,Z 1004.755,A 0.000,B 0.000,C 90.000,E1 351.894} C_DIS
LIN {X -0.028,Y -554.931,Z 1004.752,A 0.000,B 0.000,C 90.000,E1 351.319} C_DIS
LIN {X -0.026,Y -560.571,Z 1004.748,A 0.000,B 0.000,C 90.000,E1 350.622} C_DIS
LIN {X 0.274,Y -564.737,Z 1004.745,A 0.000,B 0.000,C 90.000,E1 350.038} C_DIS
LIN {X -0.194,Y -569.242,Z 1004.741,A 0.000,B 0.000,C 90.000,E1 349.398} C_DIS
LIN {X 0.130,Y -574.940,Z 1004.736,A 0.000,B 0.000,C 90.000,E1 348.409} C_DIS
LIN {X 0.191,Y -579.408,Z 1004.731,A 0.000,B 0.000,C 90.000,E1 347.589} C_DIS
LIN {X 0.100,Y -584.866,Z 1004.725,A 0.000,B 0.000,C 90.000,E1 346.520} C_DIS
LIN {X -0.134,Y -590.615,Z 1004.719,A 0.000,B 0.000,C 90.000,E1 345.338} C_DIS
LIN {X 0.011,Y -594.833,Z 1004.713,A 0.000,B 0.000,C 90.000,E1 344.393} C_DIS
LIN {X -0.082,Y -597.703,Z 1004.710,A 0.000,B 0.000,C 90.000,E1 343.740} C_DIS
LIN {X -0.030,Y -603.136,Z 1004.702,A 0.000,B 0.000,C 90.000,E1 342.417} C_DIS
LIN {X -0.104,Y -606.261,Z 1004.698,A 0.000,B 0.000,C 90.000,E1 341.638} C_DIS
LIN {X -0.220,Y -610.240,Z 1004.692,A 0.000,B 0.000,C 90.000,E1 340.604} C_DIS
LIN {X 0.031,Y -612.177,Z 1004.689,A 0.000,B 0.000,C 90.000,E1 340.061} C_DIS
LIN {X -0.010,Y -615.558,Z 1004.684,A 0.000,B 0.000,C 90.000,E1 339.028} C_DIS
LIN {X -0.058,Y -620.232,Z 1004.675,A 0.000,B 0.000,C 90.000,E1 337.486} C_DIS
LIN {X 0.230,Y -623.881,Z 1004.668,A 0.000,B 0.000,C 90.000,E1 336.177} C_DIS
LIN {X 0.007,Y -627.114,Z 1004.661,A 0.000,B 0.000,C 90.000,E1 334.921} C_DIS
LIN {X 0.104,Y -630.089,Z 1004.654,A 0.000,B 0.000,C 90.000,E1 333.640} C_DIS
LIN {X 0.190,Y -631.697,Z 1004.649,A 0.000,B 0.000,C 90.000,E1 332.871} C_DIS
LIN {X -0.196,Y -634.115,Z 1004.642,A 0.000,B 0.000,C 90.000,E1 331.641} C_DIS
LIN {X -0.192,Y -636.696,Z 1004.634,A 0.000,B 0.000,C 90.000,E1 330.127} C_DIS
LIN {X -0.237,Y -638.298,Z 1004.628,A 0.000,B 0.000,C 90.000,E1 329.125} C_DIS
LIN {X -0.260,Y -639.699,Z 1004.623,A 0.000,B 0.000,C 90.000,E1 328.122} C_DIS
LIN {X -0.270,Y -640.925,Z 1004.617,A 0.000,B 0.000,C 90.000,E1 327.120} C_DIS
LIN {X -0.409,Y -642.230,Z 1004.610,A 0.000,B 0.000,C 90.000,E1 325.881} C_DIS
LIN {X -0.046,Y -643.089,Z 1004.605,A 0.000,B 0.000,C 90.000,E1 324.848} C_DIS
LIN {X -0.305,Y -643.762,Z 1004.598,A 0.000,B 0.000,C 90.000,E1 323.623} C_DIS
LIN {X -0.126,Y -644.413,Z 1004.589,A 0.000,B 0.000,C 90.000,E1 322.110} C_DIS
LIN {X -0.027,Y -644.979,Z 1004.580,A 0.000,B 0.000,C 90.000,E1 320.356} C_DIS
LIN {X -0.299,Y -646.485,Z 1004.563,A 0.000,B 0.000,C 90.000,E1 317.391} C_DIS
LIN {X -0.217,Y -647.266,Z 1004.555,A 0.000,B 0.000,C 90.000,E1 315.891} C_DIS
LIN {X 0.335,Y -648.122,Z 1004.547,A 0.000,B 0.000,C 90.000,E1 314.352} C_DIS
LIN {X 0.040,Y -648.985,Z 1004.540,A 0.000,B 0.000,C 90.000,E1 313.137} C_DIS
LIN {X -0.272,Y -649.923,Z 1004.531,A 0.000,B 0.000,C 90.000,E1 311.676} C_DIS
LIN {X -0.011,Y -650.654,Z 1004.525,A 0.000,B 0.000,C 90.000,E1 310.415} C_DIS
LIN {X 0.143,Y -651.368,Z 1004.515,A 0.000,B 0.000,C 90.000,E1 308.669} C_DIS
LIN {X 0.022,Y -651.856,Z 1004.508,A 0.000,B 0.000,C 90.000,E1 307.443} C_DIS
LIN {X -0.015,Y -652.129,Z 1004.503,A 0.000,B 0.000,C 90.000,E1 306.457} C_DIS
LIN {X -0.041,Y -652.288,Z 1004.497,A 0.000,B 0.000,C 90.000,E1 305.471} C_DIS
LIN {X -0.010,Y -652.773,Z 1004.485,A 0.000,B 0.000,C 90.000,E1 303.245} C_DIS
LIN {X -0.182,Y -656.152,Z 1004.460,A 0.000,B 0.000,C 90.000,E1 298.821} C_DIS
LIN {X 0.202,Y -658.708,Z 1004.449,A 0.000,B 0.000,C 90.000,E1 296.821} C_DIS
LIN {X 0.252,Y -660.435,Z 1004.442,A 0.000,B 0.000,C 90.000,E1 295.591} C_DIS
LIN {X -0.099,Y -661.683,Z 1004.437,A 0.000,B 0.000,C 90.000,E1 294.643} C_DIS
LIN {X 0.033,Y -662.487,Z 1004.433,A 0.000,B 0.000,C 90.000,E1 293.898} C_DIS
LIN {X -0.297,Y -663.174,Z 1004.427,A 0.000,B 0.000,C 90.000,E1 292.950} C_DIS
LIN {X -0.283,Y -663.389,Z 1004.425,A 0.000,B 0.000,C 90.000,E1 292.461} C_DIS
LIN {X -0.149,Y -663.456,Z 1004.423,A 0.000,B 0.000,C 90.000,E1 292.206} C_DIS
LIN {X -0.016,Y -663.387,Z 1004.422,A 0.000,B 0.000,C 90.000,E1 291.950} C_DIS
LIN {X 0.000,Y -662.968,Z 1004.419,A 0.000,B 0.000,C 90.000,E1 291.461} C_DIS
LIN {X 0.015,Y -661.861,Z 1004.417,A 0.000,B 0.000,C 90.000,E1 290.972} C_DIS
LIN {X -0.096,Y -661.019,Z 1004.415,A 0.000,B 0.000,C 90.000,E1 290.737} C_DIS
LIN {X 0.026,Y -659.412,Z 1004.414,A 0.000,B 0.000,C 90.000,E1 290.482} C_DIS
LIN {X -0.035,Y -656.795,Z 1004.412,A 0.000,B 0.000,C 90.000,E1 290.120} C_DIS
LIN {X 0.018,Y -655.558,Z 1004.411,A 0.000,B 0.000,C 90.000,E1 289.993} C_DIS
LIN {X -0.147,Y -649.040,Z 1004.409,A 0.000,B 0.000,C 90.000,E1 289.577} C_DIS
LIN {X -0.034,Y -641.436,Z 1004.406,A 0.000,B 0.000,C 90.000,E1 289.141} C_DIS
LIN {X 0.309,Y -635.339,Z 1004.405,A 0.000,B 0.000,C 90.000,E1 288.779} C_DIS
LIN {X -0.295,Y -634.194,Z 1004.404,A 0.000,B 0.000,C 90.000,E1 288.725} C_DIS
LIN {X -0.336,Y -634.172,Z 1004.404,A 0.000,B 0.000,C 90.000,E1 288.725} C_DIS
LIN {X -0.088,Y -634.578,Z 1004.403,A 0.000,B 0.000,C 90.000,E1 288.489} C_DIS
LIN {X 0.020,Y -635.916,Z 1004.401,A 0.000,B 0.000,C 90.000,E1 288.236} C_DIS
LIN {X -0.163,Y -637.515,Z 1004.400,A 0.000,B 0.000,C 90.000,E1 288.000} C_DIS
LIN {X -0.331,Y -639.850,Z 1004.398,A 0.000,B 0.000,C 90.000,E1 287.638} C_DIS
LIN {X 0.111,Y -641.614,Z 1004.396,A 0.000,B 0.000,C 90.000,E1 287.347} C_DIS
LIN {X -0.039,Y -646.115,Z 1004.392,A 0.000,B 0.000,C 90.000,E1 286.622} C_DIS
LIN {X -0.310,Y -649.445,Z 1004.389,A 0.000,B 0.000,C 90.000,E1 286.024} C_DIS
LIN {X 0.071,Y -652.067,Z 1004.385,A 0.000,B 0.000,C 90.000,E1 285.371} C_DIS
LIN {X -0.180,Y -653.827,Z 1004.383,A 0.000,B 0.000,C 90.000,E1 284.898} C_DIS
LIN {X -0.135,Y -654.609,Z 1004.381,A 0.000,B 0.000,C 90.000,E1 284.647} C_DIS
LIN {X 0.262,Y -655.786,Z 1004.379,A 0.000,B 0.000,C 90.000,E1 284.120} C_DIS
LIN {X -0.078,Y -657.114,Z 1004.375,A 0.000,B 0.000,C 90.000,E1 283.411} C_DIS
LIN {X 0.233,Y -657.770,Z 1004.370,A 0.000,B 0.000,C 90.000,E1 282.647} C_DIS
LIN {X 0.015,Y -657.972,Z 1004.368,A 0.000,B 0.000,C 90.000,E1 282.175} C_DIS
LIN {X -0.337,Y -657.975,Z 1004.365,A 0.000,B 0.000,C 90.000,E1 281.715} C_DIS
LIN {X 0.091,Y -657.729,Z 1004.362,A 0.000,B 0.000,C 90.000,E1 281.186} C_DIS
LIN {X -0.363,Y -656.912,Z 1004.358,A 0.000,B 0.000,C 90.000,E1 280.489} C_DIS
LIN {X 0.055,Y -656.058,Z 1004.355,A 0.000,B 0.000,C 90.000,E1 279.962} C_DIS
LIN {X -0.293,Y -654.938,Z 1004.353,A 0.000,B 0.000,C 90.000,E1 279.500} C_DIS
LIN {X 0.107,Y -653.456,Z 1004.350,A 0.000,B 0.000,C 90.000,E1 278.973} C_DIS
LIN {X -0.254,Y -651.614,Z 1004.347,A 0.000,B 0.000,C 90.000,E1 278.511} C_DIS
LIN {X 0.255,Y -650.587,Z 1004.346,A 0.000,B 0.000,C 90.000,E1 278.219} C_DIS
LIN {X -0.120,Y -648.221,Z 1004.343,A 0.000,B 0.000,C 90.000,E1 277.757} C_DIS
LIN {X 0.010,Y -644.317,Z 1004.340,A 0.000,B 0.000,C 90.000,E1 277.125} C_DIS
LIN {X 0.236,Y -640.581,Z 1004.337,A 0.000,B 0.000,C 90.000,E1 276.606} C_DIS
LIN {X -0.260,Y -635.149,Z 1004.333,A 0.000,B 0.000,C 90.000,E1 276.024} C_DIS
LIN {X -0.126,Y -630.248,Z 1004.331,A 0.000,B 0.000,C 90.000,E1 275.511} C_DIS
LIN {X 0.208,Y -625.068,Z 1004.328,A 0.000,B 0.000,C 90.000,E1 274.992} C_DIS
LIN {X 0.166,Y -619.645,Z 1004.325,A 0.000,B 0.000,C 90.000,E1 274.531} C_DIS
LIN {X -0.103,Y -612.181,Z 1004.322,A 0.000,B 0.000,C 90.000,E1 274.012} C_DIS
LIN {X 0.162,Y -604.229,Z 1004.320,A 0.000,B 0.000,C 90.000,E1 273.498} C_DIS
LIN {X 0.281,Y -599.417,Z 1004.318,A 0.000,B 0.000,C 90.000,E1 273.212} C_DIS
LIN {X -0.201,Y -592.414,Z 1004.316,A 0.000,B 0.000,C 90.000,E1 272.922} C_DIS
LIN {X 0.037,Y -588.592,Z 1004.315,A 0.000,B 0.000,C 90.000,E1 272.751} C_DIS
LIN {X -0.157,Y -584.890,Z 1004.315,A 0.000,B 0.000,C 90.000,E1 272.636} C_DIS
LIN {X -0.057,Y -577.320,Z 1004.313,A 0.000,B 0.000,C 90.000,E1 272.407} C_DIS
LIN {X -0.270,Y -571.922,Z 1004.313,A 0.000,B 0.000,C 90.000,E1 272.293} C_DIS
LIN {X 0.229,Y -564.800,Z 1004.312,A 0.000,B 0.000,C 90.000,E1 272.121} C_DIS
LIN {X -0.241,Y -558.491,Z 1004.312,A 0.000,B 0.000,C 90.000,E1 272.121} C_DIS
LIN {X -0.275,Y -543.198,Z 1004.312,A 0.000,B 0.000,C 90.000,E1 272.121} C_DIS
LIN {X 0.222,Y -542.425,Z 1004.308,A 0.000,B 0.000,C 90.000,E1 271.489} C_DIS
LIN {X -0.113,Y -540.821,Z 1004.296,A 0.000,B 0.000,C 90.000,E1 269.255} C_DIS
LIN {X 0.008,Y -539.906,Z 1004.288,A 0.000,B 0.000,C 90.000,E1 267.822} C_DIS
LIN {X 0.167,Y -538.411,Z 1004.277,A 0.000,B 0.000,C 90.000,E1 265.812} C_DIS
LIN {X 0.278,Y -537.258,Z 1004.269,A 0.000,B 0.000,C 90.000,E1 264.375} C_DIS
LIN {X -0.112,Y -536.043,Z 1004.261,A 0.000,B 0.000,C 90.000,E1 262.989} C_DIS
LIN {X 0.008,Y -534.684,Z 1004.253,A 0.000,B 0.000,C 90.000,E1 261.546} C_DIS
LIN {X 0.175,Y -533.208,Z 1004.245,A 0.000,B 0.000,C 90.000,E1 260.095} C_DIS
LIN {X -0.134,Y -531.032,Z 1004.234,A 0.000,B 0.000,C 90.000,E1 258.117} C_DIS
LIN {X 0.168,Y -529.497,Z 1004.226,A 0.000,B 0.000,C 90.000,E1 256.645} C_DIS
LIN {X -0.095,Y -528.217,Z 1004.220,A 0.000,B 0.000,C 90.000,E1 255.519} C_DIS
LIN {X -0.022,Y -525.637,Z 1004.207,A 0.000,B 0.000,C 90.000,E1 253.196} C_DIS
LIN {X -0.191,Y -524.037,Z 1004.199,A 0.000,B 0.000,C 90.000,E1 251.764} C_DIS
LIN {X -0.219,Y -522.620,Z 1004.192,A 0.000,B 0.000,C 90.000,E1 250.604} C_DIS
LIN {X -0.141,Y -520.371,Z 1004.182,A 0.000,B 0.000,C 90.000,E1 248.847} C_DIS
LIN {X -0.033,Y -518.879,Z 1004.176,A 0.000,B 0.000,C 90.000,E1 247.667} C_DIS
LIN {X 0.057,Y -517.333,Z 1004.169,A 0.000,B 0.000,C 90.000,E1 246.485} C_DIS
LIN {X 0.244,Y -514.308,Z 1004.158,A 0.000,B 0.000,C 90.000,E1 244.409} C_DIS
LIN {X 0.004,Y -511.465,Z 1004.148,A 0.000,B 0.000,C 90.000,E1 242.666} C_DIS
LIN {X -0.294,Y -508.617,Z 1004.138,A 0.000,B 0.000,C 90.000,E1 240.923} C_DIS
LIN {X 0.323,Y -506.567,Z 1004.132,A 0.000,B 0.000,C 90.000,E1 239.665} C_DIS
LIN {X 0.093,Y -503.784,Z 1004.123,A 0.000,B 0.000,C 90.000,E1 238.201} C_DIS
LIN {X 0.072,Y -500.798,Z 1004.115,A 0.000,B 0.000,C 90.000,E1 236.707} C_DIS
LIN {X 0.138,Y -496.817,Z 1004.105,A 0.000,B 0.000,C 90.000,E1 234.895} C_DIS
LIN {X -0.143,Y -493.166,Z 1004.097,A 0.000,B 0.000,C 90.000,E1 233.417} C_DIS
LIN {X 0.005,Y -487.223,Z 1004.083,A 0.000,B 0.000,C 90.000,E1 230.964} C_DIS
LIN {X -0.059,Y -484.337,Z 1004.076,A 0.000,B 0.000,C 90.000,E1 229.747} C_DIS
